		ELSE	// The transfer mode can be used as the ValveStatus is not RUNNING		
			IF iRecValveMode <> 63 AND xUploadDone = FALSE THEN	// The transfer mode is currently not active and the value is not uploaded yet
				// check whether the WebConfig blocks the access to transfer mode
				fbReadBitsFromWord(wData := awBusDataFromVTEM[0], iStartBit := 8, iEndBit := 15, iValue =>iAppStatus);
				IF iRecValveMode = 61 AND iAppStatus = 10 THEN 		// access denied by WebConfig
					xUploadError := TRUE; 
					iUploadedValue := 0; 
					iResponse := eTransferResponse.access_denied_WebConfig; 
					iCommandNumber := 3; 			// do nothing (here: command 'stop')
				ELSIF iRecValveMode = 61 AND iAppStatus = 11 THEN 	// access denied due to an active saving process
					xUploadError := TRUE; 
					iUploadedValue := 0; 
					iResponse := eTransferResponse.access_denied_saving; 
					iCommandNumber := 3; 			// do nothing (here: command 'stop')
				ELSIF iRecValveMode = 61 AND iAppStatus = 15  THEN 	// no valve detected (used value not accessible without a valve)
					xUploadError := TRUE; 
					iUploadedValue := 0; 
					iResponse := eTransferResponse.no_valve_detected; 
					iCommandNumber := 1; 			// keep uploading (here: command 'upload') In a Firmware older than 4.16(E) an empty valve keep sending ValveMode 61 and AppStatus 15. In Firmware 4.16(E) the message changes with a tranfer
				ELSIF iRecValveMode = 61 AND iAppStatus = 0 AND xTransferComplete = TRUE THEN
					// The value is uploaded and the transfer mode has been closed properly
					xUploadDone := TRUE;
					xUploadError := FALSE;
					iCommandNumber := 3; 			// command 'stop' to remain the valve stopped
				ELSE	// ready to start the transfer Channel. 
					iResponse := eTransferResponse.transferring;
					xUploadError := FALSE;
					iCommandNumber := 1; 			// command 'upload' for the value
				END_IF
				
			ELSIF iRecValveMode = 63 AND xUploadDone = FALSE THEN	// The transfer mode is active, but the value is not uploaded yet
				fbReadBitsFromWord(wData := awBusDataFromVTEM[0], iStartBit := 8, iEndBit := 12, iValue =>iRecChannel);
				fbReadBitsFromWord(wData := awBusDataFromVTEM[0], iStartBit := 13, iEndBit := 15, iValue =>iRecTransferCtrl);
				fbReadBitsFromWord(wData := awBusDataFromVTEM[1], iStartBit := 0, iEndBit := 7, iValue =>iRecAddressedTarget);
				fbReadBitsFromWord(wData := awBusDataFromVTEM[1], iStartBit := 8, iEndBit := 15, iValue =>iRecIndex);
				iRecUploadedValue := WORD_TO_INT(awBusDataFromVTEM[2]);
		 
				IF iChannel = iRecChannel AND iRecTransferCtrl = 2 AND iRecAddressedTarget = iAddressedTarget AND iRecIndex = iIndex THEN
				// The addressed parameter was mirrored by the Motion Terminal, the uploaded value can be used
					iUploadedValue := iRecUploadedValue;
					xUploadError := FALSE;
					xTransferComplete := TRUE;
					// notice the last uploaded parameter
					iLastChannel := iChannel;
					iLastAddressedTarget := iAddressedTarget;
					iLastIndex := iIndex;
													
					iCommandNumber := 2; 			// exit transfer mode
					iResponse := eTransferResponse.transfer_successful; 
				
				ELSIF iRecChannel = 0 AND iRecTransferCtrl = 0 AND iRecAddressedTarget = 0 AND iRecIndex = 0 AND iRecUploadedValue <> 0 AND xFirstCycle = FALSE THEN
					// an invalid command was sent when using the transfer Channel
					
					xUploadError := TRUE; 
					iUploadedValue := 0; 
					iCommandNumber := 1; 			// command 'upload' for the value
					
					CASE iRecUploadedValue OF	// indicates the type of the invalid command
						1: 	iResponse := eTransferResponse.invalid_Channel;
						2: 	iResponse := eTransferResponse.invalid_TransferControl;	// this should never happen. 
						3: 	iResponse := eTransferResponse.invalid_AddressedTarget;
						4: 	iResponse := eTransferResponse.invalid_Index;
						5: 	iResponse := eTransferResponse.invalid_TransferValue;	// this cannot happen with an upload
						6: 	iResponse := eTransferResponse.invalid_combination;
						7:  iResponse := eTransferResponse.access_denied_DataInUse;
						8:	iResponse := eTransferResponse.no_data_empty_slot;
					END_CASE
					
				ELSE	// A different value is treated in transfer mode or the command was mirrored wrong
					iCommandNumber := 1; 			// command 'upload' for the value
					xUploadError := FALSE;
					iResponse := eTransferResponse.transferring;
				END_IF
			
			ELSE // xUploadDone = TRUE
				IF iLastChannel = iChannel AND iLastAddressedTarget = iAddressedTarget AND iLastIndex = iIndex THEN
					// The FB is still active although the value is already uploaded
					iResponse := eTransferResponse.transfer_successful;
					xUploadError := FALSE;
					iCommandNumber := 3; 			// do nothing (here: command 'stop', MAs remain stopped)
				ELSE
					// Another value was inserted to the FB without resetting the internal state with a falling edge at xExecute before
					iResponse := eTransferResponse.FB_needs_rising_edge_xExecute;
					xUploadError := TRUE;
					iUploadedValue := 0;
					iCommandNumber := 2; 			// do nothing (here: command 'exit transfer mode')
				END_IF
			END_IF
		END_IF	
	ELSIF xInputConsistent = FALSE OR xInputValid = FALSE THEN 
		xUploadDone := FALSE;
		xUploadError := TRUE;
		IF iRecValveMode = 63 THEN
			iCommandNumber := 2; 				// command 'exit transfer mode'
		ELSE
			iCommandNumber := 3;				// command 'stop'
		END_IF
	END_IF
	
	xFirstCycle := FALSE;

ELSIF xExecute = FALSE AND xFirstCycle = FALSE THEN		// falling edge an input xExecute, resetting the function block
	IF iRecValveMode = 63 THEN
		iCommandNumber := 2;							// exit transfer mode
	ELSE
		xFirstCycle := TRUE;
		xUploadDone := FALSE;
		xUploadError := FALSE;
		xTransferComplete := FALSE;
		iResponse := eTransferResponse.ready_for_new_transfer;
		iUploadedValue := 0;
		iCommandNumber := 0;							// do nothing (idle)
	END_IF
ELSIF xExecute = FALSE AND xFirstCycle = TRUE THEN		// idle mode for the function block
	iResponse := eTransferResponse.ready_for_new_transfer;
	iCommandNumber := 0;							// do nothing (idle)
END_IF
	
CASE iCommandNumber OF
	0: // idle
	
	1: // upload the value that is addressed and specified in the input of this FB
		fbWriteValueToWord(iValue := 63, iStartBit := 0, iEndBit := 5, wDataWord := awBusDataToVTEM[0]); 				// ValveMode = 63
		fbWriteValueToWord(iValue := 0, iStartBit := 6, iEndBit := 7, wDataWord := awBusDataToVTEM[0]); 				// (empty)
		fbWriteValueToWord(iValue := iChannel, iStartBit := 8, iEndBit := 12, wDataWord := awBusDataToVTEM[0]); 		// Channel
		fbWriteValueToWord(iValue := 2, iStartBit := 13, iEndBit := 15, wDataWord := awBusDataToVTEM[0]); 				// TransferControl = upload
		fbWriteValueToWord(iValue := iAddressedTarget, iStartBit := 0, iEndBit := 7, wDataWord := awBusDataToVTEM[1]); 	// AddressedTarget
		fbWriteValueToWord(iValue := iIndex, iStartBit := 8, iEndBit := 15, wDataWord := awBusDataToVTEM[1]); 			// Index
		
		awBusDataToVTEM[2] := 0;
	
	2: // exit transfer mode
		fbWriteValueToWord(iValue := 63, iStartBit := 0, iEndBit := 5, wDataWord := awBusDataToVTEM[0]); 				// ValveMode = 63
		fbWriteValueToWord(iValue := 0, iStartBit := 6, iEndBit := 7, wDataWord := awBusDataToVTEM[0]); 				// (empty)
		fbWriteValueToWord(iValue := iChannel, iStartBit := 8, iEndBit := 12, wDataWord := awBusDataToVTEM[0]); 		// Channel
		fbWriteValueToWord(iValue := 3, iStartBit := 13, iEndBit := 15, wDataWord := awBusDataToVTEM[0]); 				// TransferControl = exit

		awBusDataToVTEM[1] := 0;
		awBusDataToVTEM[2] := 0;

	3: // stop all Motion Apps
		fbWriteValueToWord(iValue := 61, iStartBit := 0, iEndBit := 5, wDataWord := awBusDataToVTEM[0]); 				// ValveMode = 61
		fbWriteValueToWord(iValue := 0, iStartBit := 6, iEndBit := 15, wDataWord := awBusDataToVTEM[0]); 				// (empty)

		awBusDataToVTEM[1] := 0;
		awBusDataToVTEM[2] := 0;
END_CASE

END_FUNCTION_BLOCK

// Transfermode/FB_Save_Configuration_Persistent
/// This function block can be used to run the transfer mode of the Motion Terminal in order to save the complete configuration for a valve.
/// CAUTION
/// Since version 2.02 of this function block a rising edge at xExecute is needed for every single saving of the whole valve configuration

FUNCTION_BLOCK FB_Save_Configuration_Persistent
VAR_INPUT
	awBusDataFromVTEM 		: ARRAY [0..2] OF WORD; 		(* 6 bytes of process data received from the Motion Terminal *)
END_VAR

VAR_IN_OUT
	awBusDataToVTEM 		: ARRAY [0..2] OF WORD; 		(* 6 bytes of process data sent to the Motion Terminal *)
END_VAR

VAR_INPUT	
	xExecute 				: BOOL;							(* has to be set to TRUE for saving and to FALSE to reset the function block after a saving process *)
END_VAR

VAR_OUTPUT
	iResponse 				: eSavingResponse;				(* returns the status of the execution of the saving process *)
	xSavingDone 			: BOOL := FALSE; 				(* indicates whether the saving process was successful *)
	xSavingError			: BOOL := FALSE;				// indicates whether an error occurred
END_VAR

VAR
	iRecValveMode 			: INT;
	iRecValveStatus 		: eValveState;
	iCommandNumber			: INT; 							(* indicates the command to be executed *)

	fbWriteValueToWord		: FB_Write_Value_To_Word;
	fbReadBitsFromWord 		: FB_Read_Bits_From_Word;
	
	iAppStatus				: INT;
	iRecTransferCtrl		: INT;
	iRecValue				: INT;
	
	iRunningState			: INT;
	xStateChange			: BOOL;
END_VAR

(*****************************************************************************************************

Festo SE & Co. KG, Esslingen
Copyright (c) 2018. All rights reserved.

Product:            Motion Terminal VTEM
Description:        Function block to save parametrisation persistent on the Motion Terminal

Object version:     2.02
Last change:        2019-07
======================================================================================================
                                       H I S T O R Y
======================================================================================================
Version:            2.02 
Date:               2019-07        
Change/Activity:    - redesign to state machine model
                    - corrected iResponse when calling the FB for the first time with xExecute = FALSE
                    (#2510151)
					- set output xSavingDone and iResponse when the FB stops sending busdata (#2534868)
Release:            3.5.7.234
Author:             MKLP/JEBU
------------------------------------------------------------------------------------------------------
Version:            2.01
Date:               2019-05
Change/Activity:    - optimized IDLE mode (#2458151)
Release:            3.5.7.233 (CODESYS 3.5.7.2, Lib version 3.3)
Author:             JEBU
------------------------------------------------------------------------------------------------------
Version:            2.00
Date:               2019-03
Change/Activity:    - changed awBusDataToVTEM into VAR_IN_OUT (#2368965)
Release:            3.5.7.230 (CODESYS 3.5.7.2, Lib version 3.0)
Author:             JEBU
------------------------------------------------------------------------------------------------------
Version:            1.00
Date:               2017
Change/Activity:    - created
Release:            3.5.7.22 (CODESYS 3.5.7.2, Lib version 2.0)
Author:             HLBG
======================================================================================================

*****************************************************************************************************)
// read the ValveMode and the ValveState of the Motion Terminal
fbReadBitsFromWord(wData := awBusDataFromVTEM[0], iStartBit := 0, iEndBit := 5, iValue => iRecValveMode);
fbReadBitsFromWord(wData := awBusDataFromVTEM[0], iStartBit := 6, iEndBit := 7, iValue => iRecValveStatus);
// For ValveMode 61
fbReadBitsFromWord(wData := awBusDataFromVTEM[0], iStartBit := 8, iEndBit := 15, iValue => iAppStatus); 
//For ValveMode 63
fbReadBitsFromWord(wData := awBusDataFromVTEM[0], iStartBit := 13, iEndBit := 15, iValue => iRecTransferCtrl); 
iRecValue := WORD_TO_INT(awBusDataFromVTEM[2]);
//-----------------------------------------------------------------------------------------------------------
// Transition: Resetting condition when xExecute become 0 in all States except "IDLE" and "RESETTING"
	IF NOT xExecute AND iRunningState <> 10 AND iRunningState <> 100 THEN
		xStateChange := TRUE;		// Leaving current state
		iRunningState := 100;	// Choosing next state, here: RESETTING
	END_IF;
//-----------------------------------------------------------------------------------------------------------
// Local state machine
	CASE iRunningState OF
		//-----------------------------------------------------------------------------------------------------------
		// State 10: IDLE										
			10:
				//Sourcecode that is repeating every cycle in this state:
					xStateChange := FALSE;					// Indicates that this state started
					iCommandNumber := 0;					// idle					
					iResponse := eSavingResponse.ready_to_save;	
				// Transition: Next State
					IF xExecute THEN
						xStateChange := TRUE;				// Leaving this state
						iRunningState := 20;				// Choosing next state, here: STARTING
					END_IF;
		//---------------------------------------------------------------------------------------------------------
		// State 20: STARTING									
			20:
			//Sourcecode that is repeating every cycle in this state:
				xStateChange := FALSE;			// Indicates that this state started
				iResponse := eSavingResponse.preparing_to_save; 
				IF iRecValveStatus = eValveState.Running THEN						// a Motion App is running
					iCommandNumber := 3; 											// command 'stop'
				ELSIF iRecValveMode = 63 THEN
					iCommandNumber := 2;											// exit transfer mode
				END_IF;
				// Transition: Next State or "FAILURE"
					IF iRecValveMode = 61 AND iAppStatus = 10 THEN 					// access denied by WebConfig
						iResponse := eSavingResponse.access_denied_WebConfig;
						xStateChange := TRUE;										// Leaving this state
						iRunningState := 70;										// Choosing next state, here: "FAILURE-Waiting"
					ELSIF iRecValveMode = 61 AND iAppStatus = 11 THEN 				// access denied due to an active saving process on another valve
						iResponse := eSavingResponse.access_denied_saving;
						xStateChange := TRUE;											// Leaving this state
						iRunningState := 70;										// Choosing next state, here: "FAILURE-Waiting"
					ELSIF iRecValveMode = 61 AND iAppStatus = 15 THEN 				// no valve detected
						iResponse := eSavingResponse.no_valve_detected;
						xStateChange := TRUE;											// Leaving this state
						iRunningState := 70;										// Choosing next state, here: "FAILURE-Waiting"
					ELSIF iRecValveMode = 61 THEN
						xStateChange := TRUE;											// Leaving this state
						iRunningState := 30;										// Choosing next state, here: "EXECUTE"
					END_IF;	
		//---------------------------------------------------------------------------------------------------------	
		// State 30: EXECUTE - Saving
			30:
				//Sourcecode that is repeating every cycle in this state:
					xStateChange := FALSE;							// Indicates that this state started		
					iCommandNumber := 4;
					iResponse := eSavingResponse.saving_in_progress;
				// Transition: Next State or "FAILURE"
					IF iRecTransferCtrl = 4 AND iRecValveMode = 63 THEN
						IF iRecValue = 3 THEN
							iResponse := eSavingResponse.saving_not_possible;
							xStateChange := TRUE;					// Leaving this state
							iRunningState := 70;					// Choosing next state, here: "FAILURE-Waiting"
						ELSIF iRecValue = 4 THEN
							iResponse := eSavingResponse.saving_failed;
							xStateChange := TRUE;					// Leaving this state
							iRunningState := 70;					// Choosing next state, here: "FAILURE-Waiting"
						ELSIF iRecValue = 2 THEN
							xStateChange := TRUE;					// Leaving this state
							iRunningState := 50;					// Choosing next state, here: "COMPLETED"
						END_IF;
					END_IF;
		//---------------------------------------------------------------------------------------------------------	
		// State 50: COMPLETED									
			50:
				// executed only in the first cycle of this state for 1 time:
					IF xStateChange = TRUE THEN
						xStateChange := FALSE;											// Indicates that this state started
						xSavingDone := TRUE;
						iResponse := eSavingResponse.saving_successful;
					END_IF;
				//Sourcecode that is repeating every cycle in this state:
					// Transition to "FAILURE" if the Busdata changed
						IF NOT(iRecValveMode = 63 AND iRecTransferCtrl = 4 AND iRecValue = 2) THEN
							iResponse := eSavingResponse.FB_needs_rising_edge_xExecute;
							xStateChange := TRUE;										// Leaving this state
							iRunningState := 70;										// Choosing next state, here: "FAILURE-Waiting"
						END_IF; 
					// Transition to "RESETTING" is outside of the statemachine, Waiting untill xExecute is 0
		//---------------------------------------------------------------------------------------------------------
		// State 70: FAILURE								
			70:
				//Sourcecode that is repeating every cycle in this state:
					xStateChange := FALSE;					// Indicates that this state started
					xSavingError := TRUE;
					xSavingDone := FALSE;
					IF iRecValveMode = 63 THEN
						iCommandNumber := 2; 			// exit transfer mode
					ELSE
						iCommandNumber := 3;			// command 'stop' (61)
					END_IF;
				// Transition to "RESETTING" is outside of the statemachine, Waiting untill xExecute is 0
		//---------------------------------------------------------------------------------------------------------
		// State 100: RESETTING									
			100:
				//Sourcecode that is repeating every cycle in this state:
					xStateChange := FALSE;		// Indicates that this state started
					iCommandNumber := 2;
					// Transition: Back to IDLE
						IF iRecValveMode = 61 THEN
							xStateChange := TRUE;				// Leaving this state
							iRunningState := 10;			// Choosing next state, here: IDLE					
							//Resetting all Values, which need only 1 cycle to reset
								xSavingDone := FALSE;
								xSavingError := FALSE;
								iResponse := eSavingResponse.ready_to_save;
								iCommandNumber := 0; 		// ValveMode = 61
						END_IF;
		//---------------------------------------------------------------------------------------------------------
			ELSE
				xStateChange := TRUE;
				iRunningState := 10;
		//---------------------------------------------------------------------------------------------------------	
	END_CASE;
//-----------------------------------------------------------------------------------------------------------------
CASE iCommandNumber OF
	0: // IDLE

	1: 	// transfer command for a specific value
		// not provided in this FB
	
	2: // exit transfer mode
		fbWriteValueToWord(iValue := 63, iStartBit := 0, iEndBit := 5, wDataWord := awBusDataToVTEM[0]); 			// ValveMode = 63
		fbWriteValueToWord(iValue := 0, iStartBit := 6, iEndBit := 7, wDataWord := awBusDataToVTEM[0]); 			// (empty)
		fbWriteValueToWord(iValue := 0, iStartBit := 8, iEndBit := 12, wDataWord := awBusDataToVTEM[0]); 			// Channel = 0
		fbWriteValueToWord(iValue := 3, iStartBit := 13, iEndBit := 15, wDataWord := awBusDataToVTEM[0]); 			// TransferControl = exit
		awBusDataToVTEM[1] := 0;
		awBusDataToVTEM[2] := 0;

	3: // stop all MotionApps
		fbWriteValueToWord(iValue := 61, iStartBit := 0, iEndBit := 5, wDataWord := awBusDataToVTEM[0]); 			// ValveMode = 61
		fbWriteValueToWord(iValue := 0, iStartBit := 6, iEndBit := 15, wDataWord := awBusDataToVTEM[0]); 			// (empty)
		awBusDataToVTEM[1] := 0;
		awBusDataToVTEM[2] := 0;

	4: // save configuration persistent
		fbWriteValueToWord(iValue := 63, iStartBit := 0, iEndBit := 5, wDataWord := awBusDataToVTEM[0]); 			// ValveMode = 63
		fbWriteValueToWord(iValue := 0, iStartBit := 6, iEndBit := 7, wDataWord := awBusDataToVTEM[0]); 			// (empty)
		fbWriteValueToWord(iValue := 0, iStartBit := 8, iEndBit := 12, wDataWord := awBusDataToVTEM[0]); 			// Channel = 0
		fbWriteValueToWord(iValue := 4, iStartBit := 13, iEndBit := 15, wDataWord := awBusDataToVTEM[0]); 			// TransferControl = save persistent
		awBusDataToVTEM[1] := 0; 																					// AddressedTarget = Index = 0
		awBusDataToVTEM[2] := 0;																					// Value = 0
END_CASE

END_FUNCTION_BLOCK

// Transfermode/FB_Write_config_AI_Module
/// This function block can be used to download the configuration of the analog input module on the motion terminal.
/// The specific parameters of this module are the inputs of this FB and can be defined by the user. 
/// The function block uses the transfer mode to write this configuration to the Motion Terminal
/// and indicates the state of the download process.

FUNCTION_BLOCK FB_Write_config_AI_Module
VAR_INPUT
	awBusDataFromVTEM				: ARRAY [0..2] OF WORD;			// 6 bytes of process data that is received from the Motion Terminal
END_VAR

VAR_IN_OUT
	awBusDataToVTEM					: ARRAY [0..2] OF WORD;			// 6 bytes of process data that is sent to the Motion Terminal
END_VAR

VAR_INPUT
	xExecute 						: BOOL;							// has to be set to TRUE for a download and to FALSE to reset the function block after the download is done
	xAbort							: BOOL;							// Aborts the function block

	iInputModuleNr					: INT;							// Number of the input module, counted from left to right beginning with 1

	iSensorTypePort0				: INT;							// ID of the sensor type, that is connected to the port 0 (0 = no sensor, 2001 = SDAP-MHS-M50, 2002 = SDAP-MHS-M100, 2003 = SDAP-MHS-M160, 2901 = custom position sensor 1, 2902 = custom position sensor 2, 2903 = custom position sensor 3, 3001	SFAB-50U-…-2SA-…, 3002	SFAB-200U-…-2SA-…, 3003	SFAB-600U-…-2SA-…, 3004	SFAB-1000U-…-2SA-…, 3101	SFAH-50U-…-PNVBA-…, 3102	SFAH-100U-…-PNVBA-…, 3103	SFAH-200U-…-PNVBA-…, 3901	custom flow sensor 1, 3902	custom flow sensor 2, 3903	custom flow sensor 3)
	iSensorOrientPort0				: INT;							// Orientation of the sensor that is connected to the port 0 (0 = risigng current level when advancing, 1 = falling current level when advancing)
	iSensorTypePort1				: INT;							// ID of the sensor type, that is connected to the port 1 (0 = no sensor, 2001 = SDAP-MHS-M50, 2002 = SDAP-MHS-M100, 2003 = SDAP-MHS-M160, 2901 = custom position sensor 1, 2902 = custom position sensor 2, 2903 = custom position sensor 3, 3001	SFAB-50U-…-2SA-…, 3002	SFAB-200U-…-2SA-…, 3003	SFAB-600U-…-2SA-…, 3004	SFAB-1000U-…-2SA-…, 3101	SFAH-50U-…-PNVBA-…, 3102	SFAH-100U-…-PNVBA-…, 3103	SFAH-200U-…-PNVBA-…, 3901	custom flow sensor 1, 3902	custom flow sensor 2, 3903	custom flow sensor 3)
	iSensorOrientPort1				: INT;							// Orientation of the sensor that is connected to the port 1 (0 = risigng current level when advancing, 1 = falling current level when advancing)
	iSensorTypePort2				: INT;							// ID of the sensor type, that is connected to the port 2 (0 = no sensor, 2001 = SDAP-MHS-M50, 2002 = SDAP-MHS-M100, 2003 = SDAP-MHS-M160, 2901 = custom position sensor 1, 2902 = custom position sensor 2, 2903 = custom position sensor 3, 3001	SFAB-50U-…-2SA-…, 3002	SFAB-200U-…-2SA-…, 3003	SFAB-600U-…-2SA-…, 3004	SFAB-1000U-…-2SA-…, 3101	SFAH-50U-…-PNVBA-…, 3102	SFAH-100U-…-PNVBA-…, 3103	SFAH-200U-…-PNVBA-…, 3901	custom flow sensor 1, 3902	custom flow sensor 2, 3903	custom flow sensor 3)
	iSensorOrientPort2				: INT;							// Orientation of the sensor that is connected to the port 2 (0 = risigng current level when advancing, 1 = falling current level when advancing)
	iSensorTypePort3				: INT;							// ID of the sensor type, that is connected to the port 3 (0 = no sensor, 2001 = SDAP-MHS-M50, 2002 = SDAP-MHS-M100, 2003 = SDAP-MHS-M160, 2901 = custom position sensor 1, 2902 = custom position sensor 2, 2903 = custom position sensor 3, 3001	SFAB-50U-…-2SA-…, 3002	SFAB-200U-…-2SA-…, 3003	SFAB-600U-…-2SA-…, 3004	SFAB-1000U-…-2SA-…, 3101	SFAH-50U-…-PNVBA-…, 3102	SFAH-100U-…-PNVBA-…, 3103	SFAH-200U-…-PNVBA-…, 3901	custom flow sensor 1, 3902	custom flow sensor 2, 3903	custom flow sensor 3)
	iSensorOrientPort3				: INT;							// Orientation of the sensor that is connected to the port 3 (0 = risigng current level when advancing, 1 = falling current level when advancing)
	iSensorTypePort4				: INT;							// ID of the sensor type, that is connected to the port 4 (0 = no sensor, 2001 = SDAP-MHS-M50, 2002 = SDAP-MHS-M100, 2003 = SDAP-MHS-M160, 2901 = custom position sensor 1, 2902 = custom position sensor 2, 2903 = custom position sensor 3, 3001	SFAB-50U-…-2SA-…, 3002	SFAB-200U-…-2SA-…, 3003	SFAB-600U-…-2SA-…, 3004	SFAB-1000U-…-2SA-…, 3101	SFAH-50U-…-PNVBA-…, 3102	SFAH-100U-…-PNVBA-…, 3103	SFAH-200U-…-PNVBA-…, 3901	custom flow sensor 1, 3902	custom flow sensor 2, 3903	custom flow sensor 3)
	iSensorOrientPort4				: INT;							// Orientation of the sensor that is connected to the port 4 (0 = risigng current level when advancing, 1 = falling current level when advancing)
	iSensorTypePort5				: INT;							// ID of the sensor type, that is connected to the port 5 (0 = no sensor, 2001 = SDAP-MHS-M50, 2002 = SDAP-MHS-M100, 2003 = SDAP-MHS-M160, 2901 = custom position sensor 1, 2902 = custom position sensor 2, 2903 = custom position sensor 3, 3001	SFAB-50U-…-2SA-…, 3002	SFAB-200U-…-2SA-…, 3003	SFAB-600U-…-2SA-…, 3004	SFAB-1000U-…-2SA-…, 3101	SFAH-50U-…-PNVBA-…, 3102	SFAH-100U-…-PNVBA-…, 3103	SFAH-200U-…-PNVBA-…, 3901	custom flow sensor 1, 3902	custom flow sensor 2, 3903	custom flow sensor 3)
	iSensorOrientPort5				: INT;							// Orientation of the sensor that is connected to the port 5 (0 = risigng current level when advancing, 1 = falling current level when advancing)
	iSensorTypePort6				: INT;							// ID of the sensor type, that is connected to the port 6 (0 = no sensor, 2001 = SDAP-MHS-M50, 2002 = SDAP-MHS-M100, 2003 = SDAP-MHS-M160, 2901 = custom position sensor 1, 2902 = custom position sensor 2, 2903 = custom position sensor 3, 3001	SFAB-50U-…-2SA-…, 3002	SFAB-200U-…-2SA-…, 3003	SFAB-600U-…-2SA-…, 3004	SFAB-1000U-…-2SA-…, 3101	SFAH-50U-…-PNVBA-…, 3102	SFAH-100U-…-PNVBA-…, 3103	SFAH-200U-…-PNVBA-…, 3901	custom flow sensor 1, 3902	custom flow sensor 2, 3903	custom flow sensor 3)
	iSensorOrientPort6				: INT;							// Orientation of the sensor that is connected to the port 6 (0 = risigng current level when advancing, 1 = falling current level when advancing)
	iSensorTypePort7				: INT;							// ID of the sensor type, that is connected to the port 7 (0 = no sensor, 2001 = SDAP-MHS-M50, 2002 = SDAP-MHS-M100, 2003 = SDAP-MHS-M160, 2901 = custom position sensor 1, 2902 = custom position sensor 2, 2903 = custom position sensor 3, 3001	SFAB-50U-…-2SA-…, 3002	SFAB-200U-…-2SA-…, 3003	SFAB-600U-…-2SA-…, 3004	SFAB-1000U-…-2SA-…, 3101	SFAH-50U-…-PNVBA-…, 3102	SFAH-100U-…-PNVBA-…, 3103	SFAH-200U-…-PNVBA-…, 3901	custom flow sensor 1, 3902	custom flow sensor 2, 3903	custom flow sensor 3)
	iSensorOrientPort7				: INT;							// Orientation of the sensor that is connected to the port 7 (0 = risigng current level when advancing, 1 = falling current level when advancing)
END_VAR

VAR_OUTPUT
	iResponse						: eTransferResponse;			// returns the status of the execution of the download process
	sCurrentValue 					: STRING; 						// indicates which value of the array is currently treated (necessary to evaluate in case of error messages)
	xBusy							: BOOL := FALSE;				// indicates whether the function block is active 
	xDownloadDone 					: BOOL := FALSE;				// indicates whether the download was successful
	xDownloadError 					: BOOL := FALSE; 				// indicates whether an error occurred during the transfer
	xAborted						: BOOL := FALSE;				// indicates whether the function block is aborted
END_VAR

VAR
	aTransferPackages				: ARRAY [0..100] OF stTransferPackage;
	fbdownloadMultipleParameters	: FB_Download_Multiple_Parameters;
	xFirmwareValid					: BOOL := FALSE;				// TRUE if the firmware version of the motion terminal controller is at least 4.9.x
	iCurrentValue					: INT;							// Output of the function block instance of FB_Download_Multiple_Parameters
	fbWriteValueToWord 				: FB_Write_Value_To_Word;		// instance of the function block
	fbReadBitsFromWord				: FB_Read_Bits_From_Word;		// instance of the function block
	iCurrentValveModeTM				: INT;							// currently active valve mode
	iCurrentChannelTM				: INT;							// currently active channel (transfer mode)
	iCurrentAddressedTargetTM		: INT;							// currently used addressed target (transfer mode)
	iCurrentIndexTM					: INT;							// currently used index (transfer mode)
	iCurrentValueTM					: INT;							// currently used value (transfer mode)
	iCurrentFirmwareMajor			: INT;							// Major number of the firmware version actually installed in the motion terminal
	iCurrentFirmwareMinor			: INT;							// Minor number of the firmware version actually installed in the motion terminal
	iCounterMajor					: INT;							// Counter Variable for major version number timeout check
	iCounterMinor					: INT;							// Counter Variable for minor version number timeout check
	iCounterMax						: INT := 5000;					// max value for the timeout counter
	iRunningState					: INT := 10;					// currently running state of this function block
	xStateChange					: BOOL;							// TRUE if the state is changing
	iSetValveMode					: INT;
	iSetTransferControl				: INT;
	iCommandNumber					: INT;							// switch for the command case 
	iInputModuleNrFC				: INT;
	aFCTransferPackages				: ARRAY [0..100] OF stTransferPackage;
	i								: INT;
	xInputConsistent				: BOOL;
END_VAR

(*****************************************************************************************************

Festo SE & Co. KG, Esslingen
Copyright (c) 2019. All rights reserved.

Product:            Motion Terminal VTEM
Description:        Function block to download the analog module parameters to the Motion Terminal
Object version:     2.02
Last change:        2020-11
======================================================================================================
                                       H I S T O R Y
======================================================================================================
Version:            2.02
Date:               2020-11        
Change/Activity:    - added new sensor types within comments (#3760018)
Release:            3.5.7.236 (CODESYS 3.5.7.2, Lib version 3.6)
Author:             JEBU
------------------------------------------------------------------------------------------------------
Version:            2.02
Date:               2019-07        
Change/Activity:    - corrected iResponse when calling the FB for the first time with xExecute = FALSE
					(#2510151)
					- iResponse changes to "AOI_neeeds_rising_Edge_xExecute" when changing the inputs 
					  while the FB is running (#2515565)
					- iResponse changes always to "invalid_module_number" when the input iInputModuleNr
					  is wrong(#2515412)
Release:            3.5.7.234 (CODESYS 3.5.7.2, Lib version 3.4)
Author:             MKLP/JEBU
------------------------------------------------------------------------------------------------------
Version:            2.01  
Date:               2019-04        
Change/Activity:    - New States: FAILURE-Stopping and ABORTING
                    - Changed awBusDataFromVTEM into INPUT
					- renamed eResponse into iResponse
Release:            3.5.7.231 (CODESYS 3.5.7.2, Lib version 3.1)
Author:             MKLP/JEBU
------------------------------------------------------------------------------------------------------
Version:            2.00   
Date:               2019-03        
Change/Activity:    - created
Release:            3.5.7.230 (CODESYS 3.5.7.2, Lib version 3.0)
Author:             MKLP/JEBU
======================================================================================================

******************************************************************************************************)

// Read the answer from the motion terminal
	fbReadBitsFromWord(	wData:= awBusDataFromVTEM[0], iStartBit:= 0, iEndBit:= 5, iValue=> iCurrentValveModeTM, xError=> );  		// read current valve mode
	fbReadBitsFromWord(	wData:= awBusDataFromVTEM[0], iStartBit:= 8, iEndBit:= 12, iValue=> iCurrentChannelTM, 	xError=> );			// read current channel
	fbReadBitsFromWord(	wData:= awBusDataFromVTEM[1], iStartBit:= 0, iEndBit:= 7, iValue=> iCurrentAddressedTargetTM, xError=> );	// read current addressed target
	fbReadBitsFromWord(	wData:= awBusDataFromVTEM[1], iStartBit:= 8, iEndBit:= 15, iValue=> iCurrentIndexTM, xError=> );			// read current index
	fbReadBitsFromWord(	wData:= awBusDataFromVTEM[2], iStartBit:= 0, iEndBit:= 15, iValue=> iCurrentValueTM, xError=> );			// read current value
//-----------------------------------------------------------------------------------------------------------

// Transition: Aborting condition when xAbort is TRUE in all States except "IDLE" , "ABORTING", "ABORTED" and "RESETTING"
	IF xAbort = TRUE AND iRunningState <> 10 AND iRunningState <> 80 AND iRunningState <> 90 AND iRunningState <> 100 THEN
		xStateChange := TRUE;	// Leaving current state
		iRunningState := 80;	// Choosing next state, here: ABORTING
	END_IF
//-----------------------------------------------------------------------------------------------------------

// Write the Array to transfer the data
	// ID of sensor at port 0
		aTransferPackages[0].iChannel := 16;
		aTransferPackages[0].iAddressedTarget := iInputModuleNr;
		aTransferPackages[0].iIndex := 1;
		aTransferPackages[0].iTransferValue := iSensorTypePort0;
	
	// Orientation of the sensor at port 0
		aTransferPackages[1].iChannel := 16;
		aTransferPackages[1].iAddressedTarget := iInputModuleNr;
		aTransferPackages[1].iIndex := 2;
		aTransferPackages[1].iTransferValue := iSensorOrientPort0;
	
	// ID of sensor at port 1
		aTransferPackages[2].iChannel := 16;
		aTransferPackages[2].iAddressedTarget := iInputModuleNr;
		aTransferPackages[2].iIndex := 31;
		aTransferPackages[2].iTransferValue := iSensorTypePort1;
			
	// Orientation of the sensor at port 1
		aTransferPackages[3].iChannel := 16;
		aTransferPackages[3].iAddressedTarget := iInputModuleNr;
		aTransferPackages[3].iIndex := 32;
		aTransferPackages[3].iTransferValue := iSensorOrientPort1;
		
	// ID of sensor at port 2
		aTransferPackages[4].iChannel := 16;
		aTransferPackages[4].iAddressedTarget := iInputModuleNr;
		aTransferPackages[4].iIndex := 61;
		aTransferPackages[4].iTransferValue := iSensorTypePort2;
	
	// Orientation of the sensor at port 2
		aTransferPackages[5].iChannel := 16;
		aTransferPackages[5].iAddressedTarget := iInputModuleNr;
		aTransferPackages[5].iIndex := 62;
		aTransferPackages[5].iTransferValue := iSensorOrientPort2;
		
	// ID of sensor at port 3
		aTransferPackages[6].iChannel := 16;
		aTransferPackages[6].iAddressedTarget := iInputModuleNr;
		aTransferPackages[6].iIndex := 91;
		aTransferPackages[6].iTransferValue := iSensorTypePort3;
	
	// Orientation of the sensor at port 3
		aTransferPackages[7].iChannel := 16;
		aTransferPackages[7].iAddressedTarget := iInputModuleNr;
		aTransferPackages[7].iIndex := 92;
		aTransferPackages[7].iTransferValue := iSensorOrientPort3;
	
	// ID of sensor at port 4
		aTransferPackages[8].iChannel := 16;
		aTransferPackages[8].iAddressedTarget := iInputModuleNr;
		aTransferPackages[8].iIndex := 121;
		aTransferPackages[8].iTransferValue := iSensorTypePort4;
		
	// Orientation of the sensor at port 4
		aTransferPackages[9].iChannel := 16;
		aTransferPackages[9].iAddressedTarget := iInputModuleNr;
		aTransferPackages[9].iIndex := 122;
		aTransferPackages[9].iTransferValue := iSensorOrientPort4;
		
	// ID of sensor at port 5
		aTransferPackages[10].iChannel := 16;
		aTransferPackages[10].iAddressedTarget := iInputModuleNr;
		aTransferPackages[10].iIndex := 151;
		aTransferPackages[10].iTransferValue := iSensorTypePort5;
			
	// Orientation of the sensor at port 5
		aTransferPackages[11].iChannel := 16;
		aTransferPackages[11].iAddressedTarget := iInputModuleNr;
		aTransferPackages[11].iIndex := 152;
		aTransferPackages[11].iTransferValue := iSensorOrientPort5;
			
	// ID of sensor at port 6
		aTransferPackages[12].iChannel := 16;
		aTransferPackages[12].iAddressedTarget := iInputModuleNr;
		aTransferPackages[12].iIndex := 181;
		aTransferPackages[12].iTransferValue := iSensorTypePort6;
		
	// Orientation of the sensor at port 6
		aTransferPackages[13].iChannel := 16;
		aTransferPackages[13].iAddressedTarget := iInputModuleNr;
		aTransferPackages[13].iIndex := 182;
		aTransferPackages[13].iTransferValue := iSensorOrientPort6;
		
	// ID of sensor at port 7
		aTransferPackages[14].iChannel := 16;
		aTransferPackages[14].iAddressedTarget := iInputModuleNr;
		aTransferPackages[14].iIndex := 211;
		aTransferPackages[14].iTransferValue := iSensorTypePort7;
			
	// Orientation of the sensor at port 7
		aTransferPackages[15].iChannel := 16;
		aTransferPackages[15].iAddressedTarget := iInputModuleNr;
		aTransferPackages[15].iIndex := 212;
		aTransferPackages[15].iTransferValue := iSensorOrientPort7;
		
	// define end of parameter list to be downloaded by setting all variables to 0 (end criterion for FB_Download_Multiple_Parameters)
		aTransferPackages[16].iChannel := 0;
		aTransferPackages[16].iAddressedTarget := 0;
		aTransferPackages[16].iIndex := 0;
		aTransferPackages[16].iTransferValue := 0;

//-----------------------------------------------------------------------------------------------------------
// Checking if the inputs changes when the FB is not in IDLE or STARTING 
IF iRunningState = 30 OR iRunningState = 32 OR iRunningState = 34 OR iRunningState = 40 OR iRunningState = 50 OR ((iRunningState = 60 OR iRunningState = 70) AND xInputConsistent = 1) THEN
	FOR i := 0 TO 15 DO
		IF aFCTransferPackages[i].iChannel <> aTransferPackages[i].iChannel THEN
			xInputConsistent := FALSE;
		ELSIF aFCTransferPackages[i].iAddressedTarget <> aTransferPackages[i].iAddressedTarget THEN
			xInputConsistent := FALSE;
		ELSIF aFCTransferPackages[i].iIndex <> aTransferPackages[i].iIndex THEN
			xInputConsistent := FALSE;
		ELSIF aFCTransferPackages[i].iTransferValue <> aTransferPackages[i].iTransferValue THEN
			xInputConsistent := FALSE;
		END_IF;
	END_FOR;
	
	IF xInputConsistent = FALSE THEN
		iResponse := eTransferResponse.FB_needs_rising_edge_xExecute;
		xStateChange := TRUE;		// Leaving this state
		iRunningState := 60;	// Choosing next state, here: FAILURE - Stopping
	END_IF
END_IF			
//-----------------------------------------------------------------------------------------------------------

// Local state machine
	CASE iRunningState OF
		// State 10: IDLE
			10:			
			//Sourcecode that is repeating every cycle in this state:
				xStateChange := FALSE;				// Indicates that this state started
				iCommandNumber := 0;				// idle
				iResponse := eTransferResponse.ready_for_new_transfer;
			
				// Transition: Next State
					IF xExecute = TRUE THEN
						xStateChange := TRUE;		// Leaving this state
						iRunningState := 20;		// Choosing next state, here: STARTING
					END_IF
		//---------------------------------------------------------------------------------------------------------
		
		// State 20: STARTING									
			20:
			// executed only in the first cycle of this state for 1 time:
				IF xStateChange = TRUE THEN
					xStateChange := FALSE;	// Indicates that this state started
					
					//Setting local variables for a clean start				
						iCounterMajor := 1;
						iCounterMinor := 1;
						
					// store the parameter array that was given in the first cycle
						aFCTransferPackages := aTransferPackages;
						xInputConsistent := TRUE;
										
					//Setting outputs
						xBusy := TRUE;
						iResponse := eTransferResponse.reading_transfermode;
				END_IF
				
			//Sourcecode that is repeating every cycle in this state:
				//Inputs are correct: Leaving transfermode or stop motion app 
					IF iCurrentValveModeTM = 63 THEN							// exit transfer mode if transfermode is running
						iCommandNumber := 1;									// Exit Transfermode
					ELSIF iCurrentValveModeTM < 60 THEN							// stop all Motion Apps if any Motion App is running
						iCommandNumber := 2;									// Stop all Motion Apps or ValveMode = 61
					END_IF

				// Transition: Next State
					IF iCurrentValveModeTM = 61 THEN
						xStateChange := TRUE;									// Leaving this state
						iRunningState := 30;									// Choosing next state, here: Checking major firmware
					END_IF
		//---------------------------------------------------------------------------------------------------------	
		
		// State 30: EXECUTE - Checking Major Firmware			
			30:
				//Sourcecode that is repeating every cycle in this state:
					xStateChange := FALSE;	// Indicates that this state started		
		
					// check the major number of the actual version of the firmware that is installed on the motion terminal
						iCommandNumber := 3;
					
					// Transition: Next State or FAILURE
					IF iCurrentValveModeTM = 63 AND iCurrentChannelTM = 25 AND iCurrentAddressedTargetTM = 2 AND iCurrentIndexTM = 1 THEN 
						iCurrentFirmwareMajor := iCurrentValueTM;
						xStateChange := TRUE;	// Leaving this state
						iRunningState := 32;	// Choosing next state, here: Checking minor firmware and firmware compare
						
					ELSE // timeout mechanism after <iCounterMax> cycles within this state
						iCounterMajor := iCounterMajor + 1;
						IF iCounterMajor = iCounterMax THEN
							iResponse := eTransferResponse.communication_failed;
							xStateChange := TRUE;	// Leaving this state
							iRunningState := 60;	// Choosing next state, here: FAILURE - Stopping
						END_IF
					END_IF
		//---------------------------------------------------------------------------------------------------------
			
		// State 32: EXECUTE - Checking Minor Firmware			
			32:
				//Sourcecode that is repeating every cycle in this state:
					xStateChange := FALSE;	// Indicates that this state started
					
					// check the minor number of the actual version of the firmware that is installed on the motion terminal
						iCommandNumber := 4;
					
			 	// Transition: Next State or Failure(Invalid Firmware, no Response)
			 		IF iCurrentValveModeTM = 63 AND iCurrentChannelTM = 25 AND iCurrentAddressedTargetTM = 2 AND iCurrentIndexTM = 2 THEN
			 			iCurrentFirmwareMinor := iCurrentValueTM;
			 			// check firmware version >= 4.9.x
			 				IF iCurrentFirmwareMajor < 4 OR (iCurrentFirmwareMajor = 4 AND iCurrentFirmwareMinor < 9) THEN
			 					xFirmwareValid := FALSE;
			 					iResponse := eTransferResponse.invalid_firmware_version;
			 					xStateChange := TRUE;	// Leaving this state
			 					iRunningState := 60;	// Choosing next state, here: FAILURE - Stopping
			 				ELSE
			 					xFirmwareValid := 1;
			 					xStateChange := TRUE;	// Leaving this state
			 					iRunningState := 34;	// Choosing next state, here: Download Parameters
			 				END_IF
			 		ELSE // timeout mechanism after <iCounterMax> cycles within this state
			 			iCounterMinor := iCounterMinor + 1;
			 			IF iCounterMinor = iCounterMax THEN
			 				iResponse := eTransferResponse.communication_failed;
			 				xStateChange := TRUE;	// Leaving this state
			 				iRunningState := 60;	// Choosing next state, here: FAILURE - Stopping
			 			END_IF
			 		END_IF
		//---------------------------------------------------------------------------------------------------------	
		
		// State 34: EXECUTE - Download Parameters				
			34:	
			//Sourcecode that is repeating every cycle in this state:
				xStateChange := 0; // Indicates that this state started
				iCommandNumber := 0; // IDLE or Download_Multiple_Parameters is active
									
				// call the function block for multiple parameter download
					fbdownloadMultipleParameters(
							awBusDataFromVTEM:= awBusDataFromVTEM, 
							awBusDataToVTEM:= awBusDataToVTEM, 
							xExecute:= 1, 
							aTransferPackages:= aTransferPackages, 
							iResponse=> iResponse, 
							iCurrentValue=> iCurrentValue, 
							xDownloadDone=> , 
							xDownloadError=> );			
		    	
				// create output for sCurrentValue
				// The current value output is needed if there is any invalid value in order to address it correctly.
				// As the user doesn't work with indices in this function block, the current value is transformed to a string holding the name of the parameter.
					CASE iCurrentValue OF
						0: sCurrentValue := 'iSensorTypePort0';
						1: sCurrentValue := 'iSensorOrientPort0';
						2: sCurrentValue := 'iSensorTypePort1';
						3: sCurrentValue := 'iSensorOrientPort1';
						4: sCurrentValue := 'iSensorTypePort2';
						5: sCurrentValue := 'iSensorOrientPort2';
						6: sCurrentValue := 'iSensorTypePort3';
						7: sCurrentValue := 'iSensorOrientPort3';
						8: sCurrentValue := 'iSensorTypePort4';
						9: sCurrentValue := 'iSensorOrientPort4';
						10: sCurrentValue := 'iSensorTypePort5';
						11: sCurrentValue := 'iSensorOrientPort5';
						12: sCurrentValue := 'iSensorTypePort6';
						13: sCurrentValue := 'iSensorOrientPort6';
						14: sCurrentValue := 'iSensorTypePort7';
						15: sCurrentValue := 'iSensorOrientPort7';
						16: sCurrentValue := 'AllParametersWritten';
					END_CASE	
				
				// Transition: Next State
					IF fbdownloadMultipleParameters.xDownloadDone = TRUE THEN
						xStateChange := TRUE;	// Leaving this state
						iRunningState := 40;	// Choosing next state, here: COMPLETING
					END_IF
				// Transition: Error occured during the download
					IF fbdownloadMultipleParameters.xDownloadError = TRUE THEN
						IF iResponse = eTransferResponse.invalid_AddressedTarget THEN
							iResponse := eTransferResponse.invalid_module_number;
						END_IF
						xStateChange := TRUE;	// Leaving this state
						iRunningState := 60;	// Choosing next state, here: FAILURE - Stopping
					END_IF
		//---------------------------------------------------------------------------------------------------------
			
		// State 40: COMPLETING									
			40:
				//Sourcecode that is repeating every cycle in this state:
					xStateChange := FALSE;	// Indicates that this state started
					// exit transfer mode
						iCommandNumber := 1;	// Exit Transfermode
							
				// Transition: Next State
					IF iCurrentValveModeTM = 61 THEN
						xStateChange := TRUE;	// Leaving this state
						iRunningState := 50;	// Choosing next state, here: COMPLETED
					END_IF	
		//---------------------------------------------------------------------------------------------------------
		
		// State 50: COMPLETED									
			50:
				// executed only in the first cycle of this state for 1 time:
					IF xStateChange = TRUE THEN
						xStateChange := FALSE;	// Indicates that this state started
						// Changing outputs
							xBusy := FALSE;
							xDownloadDone := TRUE;
							xDownloadError := FALSE;																		
					END_IF
				//Sourcecode that is repeating every cycle in this state:
					iCommandNumber := 2;	// Stop all Motion Apps or ValveMode = 61
									
					// Transition: RESETTING, Waiting untill xExecute is FALSE
						IF xExecute = FALSE THEN
							xStateChange := TRUE;	// Leaving this state
							iRunningState := 100;	// Choosing next state, here: RESETTING
						END_IF
		//---------------------------------------------------------------------------------------------------------
					
		// State 60: FAILURE - Stopping									
			60:
				//Sourcecode that is repeating every cycle in this state:
					xStateChange := FALSE;	// Indicates that this state started
					// exit transfer mode
						iCommandNumber := 1;	// Exit Transfermode
							
				// Transition: Next State
					IF iCurrentValveModeTM = 61 THEN
						xStateChange := TRUE;	// Leaving this state
						iRunningState := 70;	// Choosing next state, here: Failure - Waiting
					END_IF	
		//---------------------------------------------------------------------------------------------------------
		
		// State 70: FAILURE - Waiting								
			70:
				// executed only in the first cycle of this state for 1 time:
					IF xStateChange = TRUE THEN
						xStateChange := FALSE;	// Indicates that this state started							
						// Changing outputs
							xBusy := FALSE;
							xDownloadError := TRUE;
							xDownloadDone := FALSE;	
					END_IF
				//Sourcecode that is repeating every cycle in this state:	
					iCommandNumber := 2;	// Stop all Motion Apps or ValveMode = 61
													
					// Transition: RESETTING, Waiting untill xExecute is FALSE
						IF xExecute = FALSE THEN
							xStateChange := TRUE;	// Leaving this state
							iRunningState := 100;	// Choosing next state, here: RESETTING
						END_IF
		//---------------------------------------------------------------------------------------------------------
		
		// State 80: ABORTING									
			80:
				//Sourcecode that is repeating every cycle in this state:
					xStateChange := FALSE;	// Indicates that this state started
					// exit transfer mode
						iCommandNumber := 1;	// Exit Transfermode
							
				// Transition: Next State
					IF iCurrentValveModeTM = 61 THEN
						xStateChange := TRUE;	// Leaving this state
						iRunningState := 90;	// Choosing next state, here: ABORTED
					END_IF		
		
		//---------------------------------------------------------------------------------------------------------	
		
		// State 90: ABORTED									
			90:
				// executed only in the first cycle of this state for 1 time:
					IF xStateChange = TRUE THEN
						xStateChange := FALSE;	// Indicates that this state started
						//Changing outputs
							xBusy := FALSE;
							xAborted := TRUE;
							xDownloadDone := FALSE;
							xDownloadError := FALSE;	
					END_IF
					
				//Sourcecode that is repeating every cycle in this state:
					iCommandNumber := 2;	// Stop all Motion Apps or ValveMode = 61
													
					// Transition: RESETTING, Waiting untill xExecute AND xABort is FALSE
						IF xExecute = FALSE AND xAbort = FALSE THEN
							xStateChange := TRUE;	// Leaving this state
							iRunningState := 100;	// Choosing next state, here: RESETTING
						END_IF
		
		//---------------------------------------------------------------------------------------------------------	
		
		// State 100: RESETTING									
			100:	
			// executed only in the first cycle of this state for 1 time:
				IF xStateChange = TRUE THEN
					xStateChange := FALSE;	// Indicates that this state started
					// Changing outputs
						xBusy := TRUE;
						iResponse := eTransferResponse.resetting;
				END_IF
				//Sourcecode that is repeating every cycle in this state:
					// Reset the function block FB_Download_Multiple_Parameters
						fbdownloadMultipleParameters(
							awBusDataFromVTEM:= awBusDataFromVTEM, 
							awBusDataToVTEM:= awBusDataToVTEM, 
							xExecute:= FALSE, 
							aTransferPackages:= , 
							iResponse=> , 
							iCurrentValue=> , 
							xDownloadDone=> , 
							xDownloadError=> );
						
					// Transition: Back to IDLE
						IF iCurrentValveModeTM = 61 THEN
							xStateChange := TRUE;	// Leaving this state
							iRunningState := 10;	// Choosing next state, here: IDLE
													
							//Resetting all Values, which need only 1 cycle to reset
							xBusy := FALSE;
							iResponse := eTransferResponse.ready_for_new_transfer;					
							xDownloadError := FALSE;
							xDownloadDone := FALSE;
							xAborted := FALSE;
							iCurrentValue := 0;
							sCurrentValue := '';
							iCounterMajor := 0;
							iCounterMinor := 0;
							iCurrentFirmwareMajor := 0;
							iCurrentFirmwareMinor := 0;
							iCommandNumber := 2; // ValveMode = 61							
						END_IF
		//---------------------------------------------------------------------------------------------------------
			ELSE
				xStateChange := TRUE;
				iRunningState := 10;
		//---------------------------------------------------------------------------------------------------------	
	END_CASE
//---------------------------------------------------------------------------------------------------------	

CASE iCommandNumber OF
	0: // IDLE or Download_Multiple_Parameters is active

	1: // Exit Transfermode
		awBusDataToVTEM[0] := 63;	// ValveMode = 63
		fbWriteValueToWord(	iValue := 3, iStartBit := 13, iEndBit := 15, wDataWord := awBusDataToVTEM[0]); // TransferControl = exit (3)
		awBusDataToVTEM[1] := 0;
		awBusDataToVTEM[2] := 0;
	
	2: // Stop all Motion Apps or ValveMode = 61
		awBusDataToVTEM[0] := 61; // ValveMode = 61
		awBusDataToVTEM[1] := 0;
		awBusDataToVTEM[2] := 0;
		
	3: // Upload major FirmwareNr
		awBusDataToVTEM[0] := 0;
		awBusDataToVTEM[1] := 0;
		awBusDataToVTEM[2] := 0;
		// check the major number of the actual version of the firmware that is installed on the motion terminal
			fbWriteValueToWord(	iValue:= 63, iStartBit:= 0, iEndBit:= 5, wDataWord:= awBusDataToVTEM[0], xError=> );		// Start transfer mode
			fbWriteValueToWord( iValue:= 25, iStartBit:= 8, iEndBit:= 12, wDataWord:= awBusDataToVTEM[0], xError=> );		// info channel	
			fbWriteValueToWord(	iValue:= 2, iStartBit:= 13, iEndBit:= 15, wDataWord:= awBusDataToVTEM[0], xError=> );		// transfer control: upload
			fbWriteValueToWord(	iValue:= 2, iStartBit:= 0, iEndBit:= 7, wDataWord:= awBusDataToVTEM[1], xError=> );			// addressed target: 2 (Software Info)
			fbWriteValueToWord(	iValue:= 1, iStartBit:= 8, iEndBit:= 15, wDataWord:= awBusDataToVTEM[1], xError=> );		// index: 1 (firmware version Controller, major number)
		
	4: // Upload minor FirmwareNr
		awBusDataToVTEM[0] := 0;
		awBusDataToVTEM[1] := 0;
		awBusDataToVTEM[2] := 0;
		// check the minor number of the actual version of the firmware that is installed on the motion terminal
			fbWriteValueToWord( iValue:= 63, iStartBit:= 0, iEndBit:= 5, wDataWord:= awBusDataToVTEM[0], xError=> );		// Start transfer mode
			fbWriteValueToWord(	iValue:= 25, iStartBit:= 8, iEndBit:= 12, wDataWord:= awBusDataToVTEM[0], xError=> );		// info channel
			fbWriteValueToWord(	iValue:= 2, iStartBit:= 13, iEndBit:= 15, wDataWord:= awBusDataToVTEM[0], xError=> );		// transfer control: upload
			fbWriteValueToWord(	iValue:= 2, iStartBit:= 0, iEndBit:= 7, wDataWord:= awBusDataToVTEM[1], xError=> );			// addressed target: 2 (Software Info)
			fbWriteValueToWord(	iValue:= 2, iStartBit:= 8, iEndBit:= 15, wDataWord:= awBusDataToVTEM[1], xError=> );		// index: 2 (firmware version Controller, minor number)
END_CASE

END_FUNCTION_BLOCK

// Transfermode/FB_Write_config_DI_Module
/// This function block can be used to download the configuration of the digital input module on the motion terminal.
/// The specific parameters of this module are the inputs of this FB and can be defined by the user. 
/// The function block uses the transfer mode to write this configuration to the Motion Terminal
/// and indicates the state of the download process.

FUNCTION_BLOCK FB_Write_config_DI_Module
VAR_INPUT
	awBusDataFromVTEM				: ARRAY [0..2] OF WORD;			// 6 bytes of process data that is received from the Motion Terminal
END_VAR

VAR_IN_OUT	
	awBusDataToVTEM					: ARRAY [0..2] OF WORD;			// 6 bytes of process data that is sent to the Motion Terminal
END_VAR

VAR_INPUT
	xExecute 						: BOOL;							// has to be set to TRUE for a download and to FALSE to reset the function block after the download is done
	xAbort							: BOOL;							// Aborts the function block

	iInputModuleNr					: INT;							// Number of the input module, counted from left to right beginning with 1

	iSensorTypePort0				: INT;							// ID of the sensor type, that is connected to the port 0 (0 = no Sensor, 1001 = SMT-8M-A-PS-24V-... (normally open contact))
	iSensorTypePort1				: INT;							// ID of the sensor type, that is connected to the port 1 (0 = no Sensor, 1001 = SMT-8M-A-PS-24V-... (normally open contact))
	iSensorTypePort2				: INT;							// ID of the sensor type, that is connected to the port 2 (0 = no Sensor, 1001 = SMT-8M-A-PS-24V-... (normally open contact))
	iSensorTypePort3				: INT;							// ID of the sensor type, that is connected to the port 3 (0 = no Sensor, 1001 = SMT-8M-A-PS-24V-... (normally open contact))
	iSensorTypePort4				: INT;							// ID of the sensor type, that is connected to the port 4 (0 = no Sensor, 1001 = SMT-8M-A-PS-24V-... (normally open contact))
	iSensorTypePort5				: INT;							// ID of the sensor type, that is connected to the port 5 (0 = no Sensor, 1001 = SMT-8M-A-PS-24V-... (normally open contact))
	iSensorTypePort6				: INT;							// ID of the sensor type, that is connected to the port 6 (0 = no Sensor, 1001 = SMT-8M-A-PS-24V-... (normally open contact))
	iSensorTypePort7				: INT;							// ID of the sensor type, that is connected to the port 7 (0 = no Sensor, 1001 = SMT-8M-A-PS-24V-... (normally open contact))
END_VAR

VAR_OUTPUT
	iResponse						: eTransferResponse;			// returns the status of the execution of the download process
	sCurrentValue 					: STRING; 						// indicates which value of the array is currently treated (necessary to evaluate in case of error messages)
	xBusy							: BOOL := FALSE;				// indicates whether the function block is active 
	xDownloadDone 					: BOOL := FALSE;				// indicates whether the download was successful
	xDownloadError 					: BOOL := FALSE; 				// indicates whether an error occurred during the transfer
	xAborted						: BOOL := FALSE;				// indicates whether the function block is aborted
END_VAR

VAR
	aTransferPackages				: ARRAY [0..100] OF stTransferPackage;
	fbdownloadMultipleParameters	: FB_Download_Multiple_Parameters;
	xFirmwareValid					: BOOL := FALSE;				// TRUE if the firmware version of the motion terminal controller is at least 4.9.x
	iCurrentValue					: INT;							// Output of the function block instance of FB_Download_Multiple_Parameters
	fbWriteValueToWord 				: FB_Write_Value_To_Word;		// instance of the function block
	fbReadBitsFromWord				: FB_Read_Bits_From_Word;		// instance of the function block
	iCurrentValveModeTM				: INT;							// currently active valve mode
	iCurrentChannelTM				: INT;							// currently active channel (transfer mode)
	iCurrentAddressedTargetTM		: INT;							// currently used addressed target (transfer mode)
	iCurrentIndexTM					: INT;							// currently used index (transfer mode)
	iCurrentValueTM					: INT;							// currently used value (transfer mode)
	iCurrentFirmwareMajor			: INT;							// Major number of the firmware version actually installed in the motion terminal
	iCurrentFirmwareMinor			: INT;							// Minor number of the firmware version actually installed in the motion terminal
	iCounterMajor					: INT;							// Counter Variable for major version number timeout check
	iCounterMinor					: INT;							// Counter Variable for minor version number timeout check
	iCounterMax						: INT := 5000;					// max value for the timeout counter
	iRunningState					: INT := 10;					// currently running state of this function block
	xStateChange					: BOOL;							// TRUE if the state is changing
	iSetValveMode					: INT;
	iSetTransferControl				: INT;
	iCommandNumber					: INT;
	aFCTransferPackages				: ARRAY [0..100] OF stTransferPackage;
	xInputConsistent				: BOOL;
	i								: INT;
END_VAR

(*****************************************************************************************************

Festo SE & Co. KG, Esslingen
Copyright (c) 2019. All rights reserved.

Product:            Motion Terminal VTEM
Description:        Function block to download the digital module parameters to the Motion Terminal
Object version:     2.02
Last change:        2019-07
======================================================================================================
                                       H I S T O R Y
======================================================================================================
Version:            2.02 
Date:               2019-07        
Change/Activity:    - corrected iResponse when calling the FB for the first time with xExecute = FALSE
					(#2510151)
					- iResponse changes to "AOI_neeeds_rising_Edge_xExecute" when changing the inputs 
					  while the FB is running (#2515565)
					- iResponse changes always to "invalid_module_number" when the input iInputModuleNr
					  is wrong(#2515412)
Release:            3.5.7.234 (CODESYS 3.5.7.2, Lib version 3.4)
Author:             MKLP/JEBU
------------------------------------------------------------------------------------------------------
Version:            2.01  
Date:               2019-04        
Change/Activity:    - New States: FAILURE-Stopping and ABORTING
                    - Changed awBusDataFromVTEM into INPUT
					- renamed eResponse into iResponse
Release:            3.5.7.231 (CODESYS 3.5.7.2, Lib version 3.1)
Author:             MKLP/JEBU
------------------------------------------------------------------------------------------------------
Version:            2.00   
Date:               2019-03        
Change/Activity:    - created
Release:            3.5.7.230 (CODESYS 3.5.7.2, Lib version 3.0)
Author:             MKLP/JEBU
======================================================================================================

******************************************************************************************************)

// Read the answer from the motion terminal
	fbReadBitsFromWord(	wData:= awBusDataFromVTEM[0], iStartBit:= 0, iEndBit:= 5, iValue=> iCurrentValveModeTM, xError=> );  		// read current valve mode
	fbReadBitsFromWord(	wData:= awBusDataFromVTEM[0], iStartBit:= 8, iEndBit:= 12, iValue=> iCurrentChannelTM, 	xError=> );			// read current channel
	fbReadBitsFromWord(	wData:= awBusDataFromVTEM[1], iStartBit:= 0, iEndBit:= 7, iValue=> iCurrentAddressedTargetTM, xError=> );	// read current addressed target
	fbReadBitsFromWord(	wData:= awBusDataFromVTEM[1], iStartBit:= 8, iEndBit:= 15, iValue=> iCurrentIndexTM, xError=> );			// read current index
	fbReadBitsFromWord(	wData:= awBusDataFromVTEM[2], iStartBit:= 0, iEndBit:= 15, iValue=> iCurrentValueTM, xError=> );			// read current value
//-----------------------------------------------------------------------------------------------------------

// Transition: Aborting condition when xAbort is TRUE in all States except "IDLE" , "ABORTING", "ABORTED" and "RESETTING"
	IF xAbort = TRUE AND iRunningState <> 10 AND iRunningState <> 80 AND iRunningState <> 90 AND iRunningState <> 100 THEN
		xStateChange := TRUE;	// Leaving current state
		iRunningState := 80;	// Choosing next state, here: ABORTING
	END_IF;
//-----------------------------------------------------------------------------------------------------------
// Write the Array to transfer the data
	// ID of sensor at port 0
		aTransferPackages[0].iChannel := 16;
		aTransferPackages[0].iAddressedTarget := iInputModuleNr;
		aTransferPackages[0].iIndex := 1;
		aTransferPackages[0].iTransferValue := iSensorTypePort0;
	
	// ID of sensor at port 1
		aTransferPackages[1].iChannel := 16;
		aTransferPackages[1].iAddressedTarget := iInputModuleNr;
		aTransferPackages[1].iIndex := 31;
		aTransferPackages[1].iTransferValue := iSensorTypePort1;
		
	// ID of sensor at port 2
		aTransferPackages[2].iChannel := 16;
		aTransferPackages[2].iAddressedTarget := iInputModuleNr;
		aTransferPackages[2].iIndex := 61;
		aTransferPackages[2].iTransferValue := iSensorTypePort2;
    
	// ID of sensor at port 3
		aTransferPackages[3].iChannel := 16;
		aTransferPackages[3].iAddressedTarget := iInputModuleNr;
		aTransferPackages[3].iIndex := 91;
		aTransferPackages[3].iTransferValue := iSensorTypePort3;
	
	// ID of sensor at port 4
		aTransferPackages[4].iChannel := 16;
		aTransferPackages[4].iAddressedTarget := iInputModuleNr;
		aTransferPackages[4].iIndex := 121;
		aTransferPackages[4].iTransferValue := iSensorTypePort4;
		
	// ID of sensor at port 5
		aTransferPackages[5].iChannel := 16;
		aTransferPackages[5].iAddressedTarget := iInputModuleNr;
		aTransferPackages[5].iIndex := 151;
		aTransferPackages[5].iTransferValue := iSensorTypePort5;
			
	// ID of sensor at port 6
		aTransferPackages[6].iChannel := 16;
		aTransferPackages[6].iAddressedTarget := iInputModuleNr;
		aTransferPackages[6].iIndex := 181;
		aTransferPackages[6].iTransferValue := iSensorTypePort6;
		
	// ID of sensor at port 7
		aTransferPackages[7].iChannel := 16;
		aTransferPackages[7].iAddressedTarget := iInputModuleNr;
		aTransferPackages[7].iIndex := 211;
		aTransferPackages[7].iTransferValue := iSensorTypePort7;
		
	// define end of parameter list to be downloaded by setting all variables to 0 (end criterion for FB_Download_Multiple_Parameters)
		aTransferPackages[8].iChannel := 0;
		aTransferPackages[8].iAddressedTarget := 0;
		aTransferPackages[8].iIndex := 0;
		aTransferPackages[8].iTransferValue := 0;

//-----------------------------------------------------------------------------------------------------------
// Checking if the inputs changes when the FB is not in IDLE or STARTING
	IF iRunningState = 30 OR iRunningState = 32 OR iRunningState = 34 OR iRunningState = 40 OR iRunningState = 50 OR ((iRunningState = 60 OR iRunningState = 70) AND xInputConsistent = 1) THEN
		FOR i := 0 TO 15 DO
			IF aFCTransferPackages[i].iChannel <> aTransferPackages[i].iChannel THEN
				xInputConsistent := FALSE;
			ELSIF aFCTransferPackages[i].iAddressedTarget <> aTransferPackages[i].iAddressedTarget THEN
				xInputConsistent := FALSE;
			ELSIF aFCTransferPackages[i].iIndex <> aTransferPackages[i].iIndex THEN
				xInputConsistent := FALSE;
			ELSIF aFCTransferPackages[i].iTransferValue <> aTransferPackages[i].iTransferValue THEN
				xInputConsistent := FALSE;
			END_IF;
		END_FOR;
		
		IF xInputConsistent = FALSE THEN
			iResponse := eTransferResponse.FB_needs_rising_edge_xExecute;
			xStateChange := 1;		// Leaving this state
			iRunningState := 60;	// Choosing next state, here: FAILURE - Stopping
		END_IF
	END_IF			
//-----------------------------------------------------------------------------------------------------------

// Local state machine
	CASE iRunningState OF
		// State 10: IDLE
			10:			
			//Sourcecode that is repeating every cycle in this state:
				xStateChange := FALSE;				// Indicates that this state started
				iCommandNumber := 0;				// idle
				iResponse := eTransferResponse.ready_for_new_transfer;
				
				// Transition: Next State
					IF xExecute = TRUE THEN
						xStateChange := TRUE;	// Leaving this state
						iRunningState := 20;	// Choosing next state, here: STARTING
					END_IF
		//---------------------------------------------------------------------------------------------------------
		
		// State 20: STARTING									
			20:
			// executed only in the first cycle of this state for 1 time:
				IF xStateChange = TRUE THEN
					xStateChange := FALSE;	// Indicates that this state started
					
					//Setting local variables for a clean start				
						iCounterMajor := 1;
						iCounterMinor := 1;
					
					// store the parameter array that was given in the first cycle
						aFCTransferPackages := aTransferPackages;
						xInputConsistent := TRUE;
						
					//Setting outputs
						xBusy := TRUE;
						iResponse := eTransferResponse.reading_transfermode;
				END_IF
				
			//Sourcecode that is repeating every cycle in this state:
				//Inputs are correct: Leaving transfermode or stop motion app 
					IF iCurrentValveModeTM = 63 THEN							// exit transfer mode if transfermode is running
						iCommandNumber := 1;									// Exit Transfermode
					ELSIF iCurrentValveModeTM < 60 THEN							// stop all Motion Apps if any Motion App is running
						iCommandNumber := 2;									// Stop all Motion Apps or ValveMode = 61
					END_IF

				// Transition: Next State 
					IF iCurrentValveModeTM = 61 THEN
						xStateChange := TRUE;									// Leaving this state
						iRunningState := 30;									// Choosing next state, here: Checking major firmware
					END_IF
		//---------------------------------------------------------------------------------------------------------	
		
		// State 30: EXECUTE - Checking Major Firmware			
			30:
				//Sourcecode that is repeating every cycle in this state:
					xStateChange := FALSE;	// Indicates that this state started		
		
					// check the major number of the actual version of the firmware that is installed on the motion terminal
						iCommandNumber := 3;
					
					// Transition: Next State or FAILURE
					IF iCurrentValveModeTM = 63 AND iCurrentChannelTM = 25 AND iCurrentAddressedTargetTM = 2 AND iCurrentIndexTM = 1 THEN 
						iCurrentFirmwareMajor := iCurrentValueTM;
						xStateChange := TRUE;	// Leaving this state
						iRunningState := 32;	// Choosing next state, here: Checking minor firmware and firmware compare
						
					ELSE // timeout mechanism after <iCounterMax> cycles within this state
						iCounterMajor := iCounterMajor + 1;
						IF iCounterMajor = iCounterMax THEN
							iResponse := eTransferResponse.communication_failed;
							xStateChange := TRUE;	// Leaving this state
							iRunningState := 60;	// Choosing next state, here: FAILURE - Stopping
						END_IF
					END_IF
		//---------------------------------------------------------------------------------------------------------
			
		// State 32: EXECUTE - Checking Minor Firmware			
			32:
				//Sourcecode that is repeating every cycle in this state:
					xStateChange := FALSE;	// Indicates that this state started
					
					// check the minor number of the actual version of the firmware that is installed on the motion terminal
						iCommandNumber := 4;
					
			 	// Transition: Next State or Failure(Invalid Firmware, no Response)
			 		IF iCurrentValveModeTM = 63 AND iCurrentChannelTM = 25 AND iCurrentAddressedTargetTM = 2 AND iCurrentIndexTM = 2 THEN
			 			iCurrentFirmwareMinor := iCurrentValueTM;
			 			// check firmware version >= 4.9.x
			 				IF iCurrentFirmwareMajor < 4 OR (iCurrentFirmwareMajor = 4 AND iCurrentFirmwareMinor < 9) THEN
			 					xFirmwareValid := FALSE;
			 					iResponse := eTransferResponse.invalid_firmware_version;
			 					xStateChange := TRUE;	// Leaving this state
			 					iRunningState := 60;	// Choosing next state, here: FAILURE
			 				ELSE
			 					xFirmwareValid := 1;
			 					xStateChange := TRUE;	// Leaving this state
			 					iRunningState := 34;	// Choosing next state, here: Download Parameters
			 				END_IF
			 		ELSE // timeout mechanism after <iCounterMax> cycles within this state
			 			iCounterMinor := iCounterMinor + 1;
			 			IF iCounterMinor = iCounterMax THEN
			 				iResponse := eTransferResponse.communication_failed;
			 				xStateChange := TRUE;	// Leaving this state
			 				iRunningState := 60;	// Choosing next state, here: FAILURE - Stopping
			 			END_IF
			 		END_IF
		//---------------------------------------------------------------------------------------------------------	
		
		// State 34: EXECUTE - Download Parameters				
			34:	
			//Sourcecode that is repeating every cycle in this state:
				xStateChange := 0; // Indicates that this state started
				
				iCommandNumber := 0; // IDLE or Download_Multiple_Parameters is active				
				// call the function block for multiple parameter download
					fbdownloadMultipleParameters(
							awBusDataFromVTEM:= awBusDataFromVTEM, 
							awBusDataToVTEM:= awBusDataToVTEM, 
							xExecute:= 1, 
							aTransferPackages:= aTransferPackages, 
							iResponse=> iResponse, 
							iCurrentValue=> iCurrentValue, 
							xDownloadDone=> , 
							xDownloadError=> );			
		    	
				// create output for sCurrentValue
				// The current value output is needed if there is any invalid value in order to address it correctly.
				// As the user doesn't work with indices in this function block, the current value is transformed to a string holding the name of the parameter.
					CASE iCurrentValue OF
						0: sCurrentValue := 'iSensorTypePort0';
						1: sCurrentValue := 'iSensorTypePort1';
						2: sCurrentValue := 'iSensorTypePort2';
						3: sCurrentValue := 'iSensorTypePort3';
						4: sCurrentValue := 'iSensorTypePort4';
						5: sCurrentValue := 'iSensorTypePort5';
						6: sCurrentValue := 'iSensorTypePort6';
						7: sCurrentValue := 'iSensorTypePort7';
						8: sCurrentValue := 'AllParametersWritten';
					END_CASE
				
				// Transition: Next State
					IF fbdownloadMultipleParameters.xDownloadDone = TRUE THEN
						xStateChange := TRUE;	// Leaving this state
						iRunningState := 40;	// Choosing next state, here: COMPLETING
					END_IF
				// Transition: Error occured during the download
					IF fbdownloadMultipleParameters.xDownloadError = TRUE THEN
						IF iResponse = eTransferResponse.invalid_AddressedTarget THEN
							iResponse := eTransferResponse.invalid_module_number;
						END_IF
						xStateChange := TRUE;	// Leaving this state
						iRunningState := 60;	// Choosing next state, here: FAILURE - Stopping
					END_IF
		//---------------------------------------------------------------------------------------------------------
			
		// State 40: COMPLETING									
			40:
				//Sourcecode that is repeating every cycle in this state:
					xStateChange := FALSE;	// Indicates that this state started
					// exit transfer mode
						iCommandNumber := 1;	// Exit Transfermode
							
				// Transition: Next State
					IF iCurrentValveModeTM = 61 THEN
						xStateChange := TRUE;	// Leaving this state
						iRunningState := 50;	// Choosing next state, here: COMPLETED
					END_IF	
		//---------------------------------------------------------------------------------------------------------
		
		// State 50: COMPLETED									
			50:
				// executed only in the first cycle of this state for 1 time:
					IF xStateChange = TRUE THEN
						xStateChange := FALSE;	// Indicates that this state started
						// Changing outputs
							xBusy := FALSE;
							xDownloadDone := TRUE;
							xDownloadError := FALSE;																		
					END_IF
				//Sourcecode that is repeating every cycle in this state:
					iCommandNumber := 2;	// Stop all Motion Apps or ValveMode = 61
					
					// Transition: RESETTING, Waiting untill xExecute is FALSE
						IF xExecute = FALSE THEN
							xStateChange := TRUE;	// Leaving this state
							iRunningState := 100;	// Choosing next state, here: RESETTING
						END_IF;
		//---------------------------------------------------------------------------------------------------------
					
		// State 60: FAILURE - Stopping									
			60:
				//Sourcecode that is repeating every cycle in this state:
					xStateChange := FALSE;	// Indicates that this state started
					// exit transfer mode
						iCommandNumber := 1;	// Exit Transfermode
							
				// Transition: Next State
					IF iCurrentValveModeTM = 61 THEN
						xStateChange := TRUE;	// Leaving this state
						iRunningState := 70;	// Choosing next state, here: Failure - Waiting
					END_IF	
		//---------------------------------------------------------------------------------------------------------
		
		// State 70: FAILURE - Waiting								
			70:
				// executed only in the first cycle of this state for 1 time:
					IF xStateChange = TRUE THEN
						xStateChange := FALSE;	// Indicates that this state started							
						// Changing outputs
							xBusy := FALSE;
							xDownloadError := TRUE;
							xDownloadDone := FALSE;	
					END_IF
				//Sourcecode that is repeating every cycle in this state:	
					iCommandNumber := 2;	// Stop all Motion Apps or ValveMode = 61
								
					// Transition: RESETTING, Waiting untill xExecute is FALSE
						IF xExecute = FALSE THEN
							xStateChange := TRUE;	// Leaving this state
							iRunningState := 100;	// Choosing next state, here: RESETTING
						END_IF;
		//---------------------------------------------------------------------------------------------------------
		
		// State 80: ABORTING									
			80:
				//Sourcecode that is repeating every cycle in this state:
					xStateChange := FALSE;	// Indicates that this state started
					// exit transfer mode
						iCommandNumber := 1;	// Exit Transfermode
							
				// Transition: Next State
					IF iCurrentValveModeTM = 61 THEN
						xStateChange := TRUE;	// Leaving this state
						iRunningState := 90;	// Choosing next state, here: ABORTED
					END_IF		
		
		//---------------------------------------------------------------------------------------------------------	
		
		// State 90: ABORTED									
			90:
				// executed only in the first cycle of this state for 1 time:
					IF xStateChange = TRUE THEN
						xStateChange := FALSE;	// Indicates that this state started
						//Changing outputs
							xBusy := FALSE;
							xAborted := TRUE;
							xDownloadDone := FALSE;
							xDownloadError := FALSE;	
					END_IF;
					
				//Sourcecode that is repeating every cycle in this state:
					iCommandNumber := 2;	// Stop all Motion Apps or ValveMode = 61
								
					// Transition: RESETTING, Waiting untill xExecute AND xABort is FALSE
						IF xExecute = FALSE AND xAbort = FALSE THEN
							xStateChange := TRUE;	// Leaving this state
							iRunningState := 100;	// Choosing next state, here: RESETTING
						END_IF;		
		
		//---------------------------------------------------------------------------------------------------------	
		
		// State 100: RESETTING									
			100:	
			// executed only in the first cycle of this state for 1 time:
				IF xStateChange = TRUE THEN
					xStateChange := FALSE;	// Indicates that this state started
					// Changing outputs
						xBusy := TRUE;
						iResponse := eTransferResponse.resetting;
				END_IF
				//Sourcecode that is repeating every cycle in this state:
					// Reset the function block FB_Download_Multiple_Parameters
						fbdownloadMultipleParameters(
							awBusDataFromVTEM:= awBusDataFromVTEM, 
							awBusDataToVTEM:= awBusDataToVTEM, 
							xExecute:= FALSE, 
							aTransferPackages:= , 
							iResponse=> , 
							iCurrentValue=> , 
							xDownloadDone=> , 
							xDownloadError=> );
						
					// Transition: Back to IDLE
						IF iCurrentValveModeTM = 61 THEN
							xStateChange := TRUE;	// Leaving this state
							iRunningState := 10;	// Choosing next state, here: IDLE
													
							//Resetting all Values, which need only 1 cycle to reset
							xBusy := FALSE;
							iResponse := eTransferResponse.ready_for_new_transfer;					
							xDownloadError := FALSE;
							xDownloadDone := FALSE;
							xAborted := FALSE;
							xInputConsistent := TRUE;
							iCurrentValue := 0;
							sCurrentValue := '';
							iCounterMajor := 0;
							iCounterMinor := 0;
							iCurrentFirmwareMajor := 0;
							iCurrentFirmwareMinor := 0;
							iCommandNumber := 2; // ValveMode = 61							
						END_IF
		//---------------------------------------------------------------------------------------------------------
			ELSE
				xStateChange := TRUE;
				xInputConsistent := TRUE;
				iRunningState := 10;
		//---------------------------------------------------------------------------------------------------------	
	END_CASE
//---------------------------------------------------------------------------------------------------------	

CASE iCommandNumber OF
	0: // IDLE or Download_Multiple_Parameters is active

	1: // Exit Transfermode
		awBusDataToVTEM[0] := 63;	// ValveMode = 63
		fbWriteValueToWord(	iValue := 3, iStartBit := 13, iEndBit := 15, wDataWord := awBusDataToVTEM[0]); // TransferControl = exit (3)
		awBusDataToVTEM[1] := 0;
		awBusDataToVTEM[2] := 0;
	
	2: // Stop all Motion Apps or ValveMode = 61
		awBusDataToVTEM[0] := 61; // ValveMode = 61
		awBusDataToVTEM[1] := 0;
		awBusDataToVTEM[2] := 0;
		
	3: // Upload major FirmwareNr
		awBusDataToVTEM[0] := 0;
		awBusDataToVTEM[1] := 0;
		awBusDataToVTEM[2] := 0;
		// check the major number of the actual version of the firmware that is installed on the motion terminal
			fbWriteValueToWord(	iValue:= 63, iStartBit:= 0, iEndBit:= 5, wDataWord:= awBusDataToVTEM[0], xError=> );		// Start transfer mode
			fbWriteValueToWord( iValue:= 25, iStartBit:= 8, iEndBit:= 12, wDataWord:= awBusDataToVTEM[0], xError=> );		// info channel	
			fbWriteValueToWord(	iValue:= 2, iStartBit:= 13, iEndBit:= 15, wDataWord:= awBusDataToVTEM[0], xError=> );		// transfer control: upload
			fbWriteValueToWord(	iValue:= 2, iStartBit:= 0, iEndBit:= 7, wDataWord:= awBusDataToVTEM[1], xError=> );			// addressed target: 2 (Software Info)
			fbWriteValueToWord(	iValue:= 1, iStartBit:= 8, iEndBit:= 15, wDataWord:= awBusDataToVTEM[1], xError=> );		// index: 1 (firmware version Controller, major number)
		
	4: // Upload minor FirmwareNr
		awBusDataToVTEM[0] := 0;
		awBusDataToVTEM[1] := 0;
		awBusDataToVTEM[2] := 0;
		// check the minor number of the actual version of the firmware that is installed on the motion terminal
			fbWriteValueToWord( iValue:= 63, iStartBit:= 0, iEndBit:= 5, wDataWord:= awBusDataToVTEM[0], xError=> );		// Start transfer mode
			fbWriteValueToWord(	iValue:= 25, iStartBit:= 8, iEndBit:= 12, wDataWord:= awBusDataToVTEM[0], xError=> );		// info channel
			fbWriteValueToWord(	iValue:= 2, iStartBit:= 13, iEndBit:= 15, wDataWord:= awBusDataToVTEM[0], xError=> );		// transfer control: upload
			fbWriteValueToWord(	iValue:= 2, iStartBit:= 0, iEndBit:= 7, wDataWord:= awBusDataToVTEM[1], xError=> );			// addressed target: 2 (Software Info)
			fbWriteValueToWord(	iValue:= 2, iStartBit:= 8, iEndBit:= 15, wDataWord:= awBusDataToVTEM[1], xError=> );		// index: 2 (firmware version Controller, minor number)
END_CASE;

END_FUNCTION_BLOCK

// Transfermode/FB_ReadMalfunctionList
/// This function block can be used to get the whole Information that is provided by the Motion Terminal inside
/// of the malfunction list. Therefore the function block changes the valve mode to Transfer Mode, reads the
/// content of the valve related malfunction list and saves it into an array of int, separated into the
/// malfunction code, subcode and classification.

FUNCTION_BLOCK FB_ReadMalfunctionList
VAR_INPUT
	awBusDataFromVTEM				: ARRAY [0..2] OF WORD;			
END_VAR

VAR_IN_OUT
	awBusDataToVTEM					: ARRAY [0..2] OF WORD;
END_VAR

VAR_INPUT
	xExecute						: BOOL;								// Must be set to TRUE in order to start the function block							
	xAbort							: BOOL;								// If TRUE the process of the function block is aborted and the function block is resetted
	usiChooseOtherValve				: USINT;							// 0 = No other valve (Valve from connected busdata is used), 100...107 = Slot 0...7 (Addressed Target 100...107) 
END_VAR

VAR_OUTPUT
	astMalfunctionlist				: ARRAY [1..40] OF stMalfunction;	// Content of the malfunction list
	iResponse						: eResponseReadMalfunctionList;		// Returns the status of the transfer process
	xBusy							: BOOL;								// TRUE if the function block executes an action
	xDone							: BOOL;								// TRUE if the content of the malfunction list was completely saved into the astMalfunctionlist
	xError							: BOOL;								// TRUE if an error occured during the process
	xAborted						: BOOL;								// TRUE if the function block was canceled by xAbort	
END_VAR

VAR
	// malfunction list variables
		iNumberOfMalfunctions		: INT;								// Number of entries in the malfunction list

	// state machine variables
		iState						: INT := 10;						// Value for the local state machine
		xStateChange				: BOOL;								// TRUE if the state is to be changed
		xStateFinished				: BOOL := FALSE;					// TRUE if the condition for changing the state is fulfilled
		iCommandNumber				: INT;								// Value for the command case

	// Current Valve variables
		iCurrentValveMode			: INT;								// 
		iCurrentValveState			: INT;								//
		iCurrentAppState			: INT;								//
		iCurrentActVal1				: INT;								//
		iCurrentActVal2				: INT;								//
		iCurrentChannelTM			: INT;								//
		iCurrentTransferControlTM	: INT;								//
		iCurrentAddressedTargetTM	: INT;								//
		iCurrentIndexTM				: INT;								//
		iCurrentValueTM				: INT;								//

	// function block instances
		fbreadbitsfromword			: FB_Read_Bits_From_Word;			//
		fbwritevaluetoword			: FB_Write_Value_To_Word;			//

	// counter variables
		iCountMFLreset				: INT;								// Counter variable for resetting the astMalfunctionlist
		iCountMFLdownload			: INT := 1;							// Counter variable for downloading the malfunctions list entries
		
	// Auxiliary variables
		usiChooseOtherValveFC		: USINT;
		xFirstTransfer				: BOOL;
		xInputConsistent			: BOOL;
END_VAR

(*****************************************************************************************************

Festo SE & Co. KG, Esslingen
Copyright (c) 2020. All rights reserved.

Product:            Motion Terminal VTEM
Description:        Function block for reading the malfunction list of a specific valve
Object version:     1.03
======================================================================================================
                                       H I S T O R Y
======================================================================================================
Version:            1.03
Date:               2020-03
Change/Activity:    - created
Release:            3.5.7.234
Author:             JEBU/MKLP
======================================================================================================

******************************************************************************************************)

// Read the current status of the the motion terminal
	fbreadbitsfromword(wData:= awBusDataFromVTEM[0], iStartBit:=0, iEndBit:= 5, iValue=> iCurrentValveMode, xError=> );				// read current valve mode
	fbreadbitsfromword(wData:= awBusDataFromVTEM[0], iStartBit:=6, iEndBit:= 7, iValue=> iCurrentValveState, xError=> );			// read current valve state

	IF iCurrentValveMode <> 63 THEN																									// Operating mode:
		fbreadbitsfromword(wData:= awBusDataFromVTEM[0], iStartBit:=8, iEndBit:= 15, iValue=> iCurrentAppState, xError=>);				// read app state
		fbreadbitsfromword(wData:= awBusDataFromVTEM[1], iStartBit:=0, iEndBit:= 15, iValue=> iCurrentActVal1, xError=>);				// read actual value 1
		fbreadbitsfromword(wData:= awBusDataFromVTEM[2], iStartBit:=0, iEndBit:= 15, iValue=> iCurrentActVal2, xError=>);				// read actual value 2
	ELSIF iCurrentValveMode = 63 THEN																								// Transfer mode:
		fbreadbitsfromword(wData:= awBusDataFromVTEM[0], iStartBit:= 8, iEndBit:= 12, iValue=> iCurrentChannelTM, xError=> );			// read current channel
		fbreadbitsfromword(wData:= awBusDataFromVTEM[0], iStartBit:= 13, iEndBit:= 15, iValue=> iCurrentTransferControlTM, xError=> );	// read current transfer 
		fbreadbitsfromword(wData:= awBusDataFromVTEM[1], iStartBit:= 0, iEndBit:= 7, iValue=> iCurrentAddressedTargetTM, xError=> );	// read current addressed target
		fbreadbitsfromword(wData:= awBusDataFromVTEM[1], iStartBit:= 8, iEndBit:= 15, iValue=> iCurrentIndexTM, xError=> );				// read current index
		fbreadbitsfromword(wData:= awBusDataFromVTEM[2], iStartBit:= 0, iEndBit:= 15, iValue=> iCurrentValueTM, xError=> );				// read current value
	END_IF
//-----------------------------------------------------------------------------------------------------------

// Transition: Aborting condition when xAbort is TRUE in all States except "IDLE" , "ABORTING" and "RESETTING"
	IF xAbort = TRUE AND NOT(iState = 10 AND xExecute = FALSE) AND iState <> 80 AND iState <> 100 THEN
		xStateChange := TRUE;	// Leaving current state
		iState := 80;	// Choosing next state, here: ABORTING

// Error: Monitoring transition for error conditions
	ELSIF (iState <> 10 AND iState <> 20 AND NOT(iState = 30 AND xFirstTransfer = FALSE AND iCurrentValveMode = 61 AND iCurrentAppState = 15) AND iState <> 70 AND iState <> 71 AND iState <> 80 AND iState <> 100) THEN		// Ignore message "no_valve_detected" in state 30 before the first Transfer
		IF iCurrentValveMode = 63 AND iCurrentChannelTM = 0 AND iCurrentTransferControlTM = 0 AND iCurrentAddressedTargetTM = 0 AND iCurrentIndexTM = 0 THEN
			xStateChange := TRUE;
			iState := 71;	// Error during transfer mode
		ELSIF iCurrentValveMode = 61 AND iCurrentAppState <> 0 THEN
			xStateChange := TRUE;
			iState := 70;	// Error
		END_IF
	
// Error for inconsistent input usiChooseOtherValve		
	ELSIF iState <> 10 AND iState <> 20 AND iState <> 80 AND iState <> 100 AND usiChooseOtherValve <> usiChooseOtherValveFC AND xInputConsistent = TRUE THEN
		xInputConsistent := FALSE;
		xStateChange := TRUE;
		iState := 70; // Error
	END_IF

//-----------------------------------------------------------------------------------------------------------

// local state machine
	CASE iState OF
		10:	// IDLE
			// code that is executed only in the first cycle of this state
				IF xStateChange = TRUE THEN
					xStateChange := FALSE;
					iResponse := eResponseReadMalfunctionList.idle;
					xDone := FALSE;
					xError := FALSE;
					xBusy := FALSE;
					xAborted := FALSE;
				END_IF
			//-----------------------------------------------------------------------------------------------------------
			
			// code that is repeated every cycle in this state
				iCommandNumber := 0;
			//-----------------------------------------------------------------------------------------------------------
			
			// Transition
			IF xExecute = TRUE THEN
				xStateChange := TRUE;
				iState := 20;
			END_IF
			//-----------------------------------------------------------------------------------------------------------
		
		20:	// RESETTING VALVE MODE TO 61
			// code that is executed only in the first cycle of this state
				IF xStateChange = TRUE THEN
					xStateChange := FALSE;
					iResponse := eResponseReadMalfunctionList.setting_valve_to_inactive;
					xDone := FALSE;
					xError := FALSE;
					xBusy := TRUE;
					xAborted := FALSE;
					usiChooseOtherValveFC := usiChooseOtherValve;
					xInputConsistent := TRUE;
				END_IF
			//-----------------------------------------------------------------------------------------------------------
			
			// code that is repeated every cycle in this state	
				IF iCurrentValveMode = 63 THEN
					iCommandNumber := 5;	// exit transfer mode
				ELSIF iCurrentValveMode <> 61 AND iCurrentValveMode <> 63 THEN
					iCommandNumber := 6;	// stop running motion apps
				END_IF 
			//-----------------------------------------------------------------------------------------------------------
			
			// Transition
				IF iCurrentValveMode = 61 THEN
					xStateChange := TRUE;	// Leave this state
					iState := 30;			
				END_IF
			//-----------------------------------------------------------------------------------------------------------
		
		30:	// GETTING NUMBER OF MALFUNCTION MESSAGES
			// code that is executed only in the first cycle of this state
				IF xStateChange = TRUE THEN
					xStateChange := FALSE;
					iResponse := eResponseReadMalfunctionList.getting_malfunction_count;
					xDone := FALSE;
					xError := FALSE;
					xBusy := TRUE;
					xAborted := FALSE;
				END_IF
			//-----------------------------------------------------------------------------------------------------------
			
			// code that is repeated every cycle in this state	
			IF iCurrentValveMode = 61 THEN
				iCommandNumber := 10;	// getting count of malfunction messages
			ELSIF iCurrentValveMode = 63 AND iCurrentChannelTM = 31 AND iCurrentTransferControlTM = 2 AND iCurrentAddressedTargetTM = usiChooseOtherValve AND iCurrentIndexTM = 255 THEN
				iNumberOfMalfunctions := WORD_TO_INT(awBusDataFromVTEM[2]);
				xStateFinished := TRUE;
			ELSIF iCurrentValveMode = 63 AND iCommandNumber = 10 THEN // First Transfer is detected when iCurrentValveMode changes from 61 to 63. The first transfer is always with iCommandNumber = 10
				xFirstTransfer := TRUE;
			END_IF
			
			//-----------------------------------------------------------------------------------------------------------
			
			// Transition
				IF xStateFinished = TRUE THEN
					IF iNumberOfMalfunctions = 0 THEN
						xStateFinished := FALSE;
						xStateChange := TRUE;
						iState := 51; // Done with empty malfunction list
					ELSE
						xStateFinished := FALSE;
						xStateChange := TRUE;
						iState := 40; // Reading malfunction list
					END_IF
				END_IF
			//-----------------------------------------------------------------------------------------------------------

		40:	// READING MALFUNCTION LIST
			// code that is executed only in the first cycle of this state
				IF xStateChange = TRUE THEN
					xStateChange := FALSE;
					iResponse := eResponseReadMalfunctionList.transferring;
					xDone := FALSE;
					xError := FALSE;
					xBusy := TRUE;
					xAborted := FALSE;
				END_IF
			//-----------------------------------------------------------------------------------------------------------
			
			// code that is repeated every cycle in this state	
				iCommandNumber := 40;
				
				WHILE iCountMFLdownload <= iNumberOfMalfunctions DO		// go trough the malfunction list, starting with the entry at position 1 up to the last entry
					
					IF iCurrentValveMode = 63 AND iCurrentChannelTM = 31 AND iCurrentTransferControlTM = 2 AND iCurrentAddressedTargetTM = usiChooseOtherValve AND iCurrentIndexTM = iCountMFLdownload THEN
						fbreadbitsfromword(wData:=awBusDataFromVTEM[2], iStartBit:=0, iEndBit:=7, iValue:= , xError:=);					// Read malfunction code
						astMalfunctionlist[iCountMFLdownload].usiMalfunctionCode := INT_TO_USINT(fbreadbitsfromword.iValue);			// Save malfunction code
						
						fbreadbitsfromword(wData:=awBusDataFromVTEM[2], iStartBit:=8, iEndBit:=13, iValue:= , xError:=);				// Read malfunction subcode
						astMalfunctionlist[iCountMFLdownload].usiMalfunctionSubcode := INT_TO_USINT(fbreadbitsfromword.iValue);			// Save malfunction subcode
						
						fbreadbitsfromword(wData:=awBusDataFromVTEM[2], iStartBit:=14, iEndBit:=15, iValue:= , xError:=);				// Read malfunction classification
						astMalfunctionlist[iCountMFLdownload].usiMalfunctionClassification := INT_TO_USINT(fbreadbitsfromword.iValue);	// Save malfunction classification
						
						IF iCountMFLdownload = iNumberOfMalfunctions THEN
							xStateFinished := TRUE;
							EXIT;
						ELSE
							iCountMFLdownload := iCountMFLdownload + 1;
						END_IF
					ELSE
						EXIT;
					END_IF
				END_WHILE
			//-----------------------------------------------------------------------------------------------------------
			
			// Transition
				IF xStateFinished = TRUE THEN
					xStateFinished := FALSE;
					xStateChange := TRUE;
					iState := 50;	// done
					iCommandNumber := 0;	// idle
				END_IF
			//-----------------------------------------------------------------------------------------------------------
			
		50:	// DONE
			// code that is executed only in the first cycle of this state
				IF xStateChange = TRUE THEN
					xStateChange := FALSE;
					iResponse := eResponseReadMalfunctionList.done;
					xDone := TRUE;
					xError := FALSE;
					xBusy := FALSE;
					xAborted := FALSE;
				END_IF
			//-----------------------------------------------------------------------------------------------------------
			
			// code that is repeated every cycle in this state	
				iCommandNumber := 5;	// exit transfer mode
			//-----------------------------------------------------------------------------------------------------------
			
			// Transition
				IF xExecute = FALSE THEN
					xStateChange := TRUE;
					iState := 100;
				END_IF
			//-----------------------------------------------------------------------------------------------------------
			
		51:	// DONE WITH EMPTY MALFUNCTION LIST
			// code that is executed only in the first cycle of this state
				IF xStateChange = TRUE THEN
					xStateChange := FALSE;
					iResponse := eResponseReadMalfunctionList.no_entries_in_malfunction_list;
					xDone := TRUE;
					xError := FALSE;
					xBusy := FALSE;
					xAborted := FALSE;
				END_IF
			//-----------------------------------------------------------------------------------------------------------
			
			// code that is repeated every cycle in this state	
				iCommandNumber := 5;	// exit transfer mode
			//-----------------------------------------------------------------------------------------------------------
			
			// Transition
				IF xExecute = FALSE THEN
					xStateChange := TRUE;
					iState := 100;
				END_IF
			//-----------------------------------------------------------------------------------------------------------
			
		70:	// ERROR
			// code that is executed only in the first cycle of this state
				IF xStateChange = TRUE THEN
					xStateChange := FALSE;
					iResponse := eResponseReadMalfunctionList.error_while_transmitting_data_to_vtem;
					xDone := FALSE;
					xError := TRUE;
					xBusy := FALSE;
					xAborted := FALSE;
				END_IF
			//-----------------------------------------------------------------------------------------------------------
				IF xInputConsistent = FALSE THEN
					iResponse := eResponseReadMalfunctionList.FB_needs_rising_edge_xExecute;
				END_IF
			
			// code that is repeated every cycle in this state	
				CASE iCurrentAppState OF
					1:	iResponse := eResponseReadMalfunctionList.invalid_SetValveMode;
					2:	iResponse := eResponseReadMalfunctionList.invalid_SetAppControl;
					3:	iResponse := eResponseReadMalfunctionList.invalid_SetAppOption;
					4:	iResponse := eResponseReadMalfunctionList.invalid_SetPointValue1;
					5:	iResponse := eResponseReadMalfunctionList.invalid_SetPointValue2;
					6:	iResponse := eResponseReadMalfunctionList.invalid_configuration;
					
					10:	iResponse := eResponseReadMalfunctionList.access_denied_WebConfig;
					11:	iResponse := eResponseReadMalfunctionList.access_denied_saving_parameterisation;
					12:	iResponse := eResponseReadMalfunctionList.no_license_for_this_MA;
					13:	iResponse := eResponseReadMalfunctionList.all_licenses_in_use;
					14:	iResponse := eResponseReadMalfunctionList.invalid_license_file;
					15:	iResponse := eResponseReadMalfunctionList.no_valve_detected;
					16:	iResponse := eResponseReadMalfunctionList.valve_self_calibration_running;
				END_CASE
			//-----------------------------------------------------------------------------------------------------------
			
			// Transition
				IF xExecute = FALSE AND xAbort = FALSE THEN
					xStateChange := TRUE;
					iState := 100;
				END_IF
			//-----------------------------------------------------------------------------------------------------------
			
		71:	// ERROR DURING TRANFER MODE
			// code that is executed only in the first cycle of this state
				IF xStateChange = TRUE THEN
					xStateChange := FALSE;
					xDone := FALSE;
					xError := TRUE;
					xBusy := FALSE;
					xAborted := FALSE;
				END_IF
			//-----------------------------------------------------------------------------------------------------------
			
			// code that is repeated every cycle in this state	
				CASE iCurrentValueTM OF
					1:	iResponse := eResponseReadMalfunctionList.invalid_Channel;
					2:	iResponse := eResponseReadMalfunctionList.invalid_TransferControl;
					3:	iResponse := eResponseReadMalfunctionList.invalid_usiChooseOtherValve; // invalid_AddtessedTarget is always invalid_usiChooseOtherValve
					4:	iResponse := eResponseReadMalfunctionList.invalid_Index;
					5:	iResponse := eResponseReadMalfunctionList.invalid_TransferValue;
					6:	iResponse := eResponseReadMalfunctionList.no_data_empty_slot;	// invalid_Combination is always no_data_empty_slot in the context of this function block
					7:	iResponse := eResponseReadMalfunctionList.access_denied_DataInUse;
					8:	iResponse := eResponseReadMalfunctionList.no_data_empty_slot;
				END_CASE
			//-----------------------------------------------------------------------------------------------------------
			
			// Transition
				IF xExecute = FALSE AND xAbort = FALSE THEN
					xStateChange := TRUE;
					iState := 100;
				END_IF
			//-----------------------------------------------------------------------------------------------------------
			
